LIN {X 0.147,Y -636.503,Z 756.613,A 0.000,B 0.000,C 90.000,E1 326.373} C_DIS
LIN {X -0.093,Y -640.964,Z 756.608,A 0.000,B 0.000,C 90.000,E1 325.515} C_DIS
LIN {X 0.327,Y -642.816,Z 756.606,A 0.000,B 0.000,C 90.000,E1 325.102} C_DIS
LIN {X 0.141,Y -649.762,Z 756.598,A 0.000,B 0.000,C 90.000,E1 323.623} C_DIS
LIN {X 0.029,Y -652.957,Z 756.594,A 0.000,B 0.000,C 90.000,E1 322.889} C_DIS
LIN {X 0.011,Y -657.013,Z 756.588,A 0.000,B 0.000,C 90.000,E1 321.904} C_DIS
LIN {X 0.017,Y -658.915,Z 756.586,A 0.000,B 0.000,C 90.000,E1 321.412} C_DIS
LIN {X -0.068,Y -663.423,Z 756.579,A 0.000,B 0.000,C 90.000,E1 320.194} C_DIS
LIN {X -0.059,Y -666.808,Z 756.573,A 0.000,B 0.000,C 90.000,E1 319.218} C_DIS
LIN {X -0.004,Y -670.699,Z 756.567,A 0.000,B 0.000,C 90.000,E1 318.000} C_DIS
LIN {X 0.105,Y -674.291,Z 756.560,A 0.000,B 0.000,C 90.000,E1 316.782} C_DIS
LIN {X 0.210,Y -676.958,Z 756.555,A 0.000,B 0.000,C 90.000,E1 315.810} C_DIS
LIN {X -0.087,Y -679.877,Z 756.548,A 0.000,B 0.000,C 90.000,E1 314.636} C_DIS
LIN {X 0.156,Y -682.512,Z 756.541,A 0.000,B 0.000,C 90.000,E1 313.419} C_DIS
LIN {X 0.366,Y -684.591,Z 756.536,A 0.000,B 0.000,C 90.000,E1 312.447} C_DIS
LIN {X 0.133,Y -686.391,Z 756.531,A 0.000,B 0.000,C 90.000,E1 311.515} C_DIS
LIN {X 0.436,Y -688.109,Z 756.525,A 0.000,B 0.000,C 90.000,E1 310.539} C_DIS
LIN {X -0.206,Y -689.467,Z 756.520,A 0.000,B 0.000,C 90.000,E1 309.644} C_DIS
LIN {X 0.137,Y -690.705,Z 756.515,A 0.000,B 0.000,C 90.000,E1 308.669} C_DIS
LIN {X 0.306,Y -692.395,Z 756.507,A 0.000,B 0.000,C 90.000,E1 307.237} C_DIS
LIN {X -0.100,Y -693.591,Z 756.500,A 0.000,B 0.000,C 90.000,E1 306.091} C_DIS
LIN {X 0.339,Y -694.977,Z 756.491,A 0.000,B 0.000,C 90.000,E1 304.405} C_DIS
LIN {X -0.203,Y -696.089,Z 756.484,A 0.000,B 0.000,C 90.000,E1 303.038} C_DIS
LIN {X 0.137,Y -697.503,Z 756.473,A 0.000,B 0.000,C 90.000,E1 301.131} C_DIS
LIN {X -0.043,Y -698.086,Z 756.468,A 0.000,B 0.000,C 90.000,E1 300.207} C_DIS
LIN {X -0.212,Y -698.422,Z 756.463,A 0.000,B 0.000,C 90.000,E1 299.283} C_DIS
LIN {X -0.201,Y -698.977,Z 756.453,A 0.000,B 0.000,C 90.000,E1 297.641} C_DIS
LIN {X -0.156,Y -699.561,Z 756.446,A 0.000,B 0.000,C 90.000,E1 296.232} C_DIS
LIN {X -0.010,Y -700.097,Z 756.440,A 0.000,B 0.000,C 90.000,E1 295.283} C_DIS
LIN {X -0.104,Y -700.180,Z 756.438,A 0.000,B 0.000,C 90.000,E1 294.823} C_DIS
LIN {X -0.127,Y -700.106,Z 756.437,A 0.000,B 0.000,C 90.000,E1 294.591} C_DIS
LIN {X -0.226,Y -699.545,Z 756.434,A 0.000,B 0.000,C 90.000,E1 294.131} C_DIS
LIN {X -0.243,Y -698.845,Z 756.433,A 0.000,B 0.000,C 90.000,E1 293.898} C_DIS
LIN {X 0.285,Y -696.516,Z 756.430,A 0.000,B 0.000,C 90.000,E1 293.387} C_DIS
LIN {X 0.138,Y -695.765,Z 756.429,A 0.000,B 0.000,C 90.000,E1 293.281} C_DIS
LIN {X -0.372,Y -694.648,Z 756.429,A 0.000,B 0.000,C 90.000,E1 293.206} C_DIS
LIN {X -0.246,Y -693.025,Z 756.428,A 0.000,B 0.000,C 90.000,E1 293.078} C_DIS
LIN {X -0.175,Y -688.248,Z 756.426,A 0.000,B 0.000,C 90.000,E1 292.770} C_DIS
LIN {X 0.245,Y -686.538,Z 756.426,A 0.000,B 0.000,C 90.000,E1 292.642} C_DIS
LIN {X -0.233,Y -683.886,Z 756.425,A 0.000,B 0.000,C 90.000,E1 292.589} C_DIS
LIN {X 0.315,Y -675.779,Z 756.424,A 0.000,B 0.000,C 90.000,E1 292.333} C_DIS
LIN {X -0.189,Y -668.158,Z 756.424,A 0.000,B 0.000,C 90.000,E1 292.259} C_DIS
LIN {X 0.079,Y -654.886,Z 756.423,A 0.000,B 0.000,C 90.000,E1 292.078} C_DIS
LIN {X 0.379,Y -645.016,Z 756.422,A 0.000,B 0.000,C 90.000,E1 291.897} C_DIS
LIN {X -0.041,Y -631.843,Z 756.420,A 0.000,B 0.000,C 90.000,E1 291.663} C_DIS
LIN {X 0.053,Y -611.303,Z 756.418,A 0.000,B 0.000,C 90.000,E1 291.153} C_DIS
LIN {X 0.063,Y -576.468,Z 756.412,A 0.000,B 0.000,C 90.000,E1 290.174} C_DIS
LIN {X 0.005,Y -565.947,Z 756.411,A 0.000,B 0.000,C 90.000,E1 289.885} C_DIS
LIN {X 0.011,Y -560.723,Z 756.409,A 0.000,B 0.000,C 90.000,E1 289.685} C_DIS
LIN {X 0.106,Y -557.840,Z 756.409,A 0.000,B 0.000,C 90.000,E1 289.523} C_DIS
LIN {X 0.033,Y -555.917,Z 756.407,A 0.000,B 0.000,C 90.000,E1 289.322} C_DIS
LIN {X -0.009,Y -555.886,Z 756.407,A 0.000,B 0.000,C 90.000,E1 289.322} C_DIS
LIN {X -0.098,Y -555.156,Z 756.406,A 0.000,B 0.000,C 90.000,E1 289.033} C_DIS
LIN {X -0.207,Y -554.525,Z 756.397,A 0.000,B 0.000,C 90.000,E1 287.511} C_DIS
LIN {X -0.264,Y -553.899,Z 756.388,A 0.000,B 0.000,C 90.000,E1 285.843} C_DIS
LIN {X -0.218,Y -553.135,Z 756.377,A 0.000,B 0.000,C 90.000,E1 283.883} C_DIS
LIN {X -0.030,Y -552.617,Z 756.368,A 0.000,B 0.000,C 90.000,E1 282.187} C_DIS
LIN {X 0.034,Y -552.142,Z 756.360,A 0.000,B 0.000,C 90.000,E1 280.782} C_DIS
LIN {X 0.079,Y -551.632,Z 756.352,A 0.000,B 0.000,C 90.000,E1 279.378} C_DIS
LIN {X 0.152,Y -550.794,Z 756.341,A 0.000,B 0.000,C 90.000,E1 277.409} C_DIS
LIN {X -0.212,Y -550.461,Z 756.337,A 0.000,B 0.000,C 90.000,E1 276.606} C_DIS
LIN {X 0.173,Y -549.687,Z 756.329,A 0.000,B 0.000,C 90.000,E1 275.163} C_DIS
LIN {X -0.060,Y -548.779,Z 756.321,A 0.000,B 0.000,C 90.000,E1 273.784} C_DIS
LIN {X 0.253,Y -547.842,Z 756.312,A 0.000,B 0.000,C 90.000,E1 272.064} C_DIS
LIN {X -0.045,Y -547.113,Z 756.304,A 0.000,B 0.000,C 90.000,E1 270.688} C_DIS
LIN {X 0.178,Y -546.162,Z 756.296,A 0.000,B 0.000,C 90.000,E1 269.255} C_DIS
LIN {X -0.076,Y -544.884,Z 756.285,A 0.000,B 0.000,C 90.000,E1 267.306} C_DIS
LIN {X 0.177,Y -543.801,Z 756.276,A 0.000,B 0.000,C 90.000,E1 265.584} C_DIS
LIN {X -0.176,Y -543.100,Z 756.269,A 0.000,B 0.000,C 90.000,E1 264.489} C_DIS
LIN {X 0.013,Y -542.093,Z 756.261,A 0.000,B 0.000,C 90.000,E1 263.053} C_DIS
LIN {X 0.238,Y -541.174,Z 756.255,A 0.000,B 0.000,C 90.000,E1 261.894} C_DIS
LIN {X -0.009,Y -539.986,Z 756.247,A 0.000,B 0.000,C 90.000,E1 260.500} C_DIS
LIN {X -0.206,Y -538.592,Z 756.238,A 0.000,B 0.000,C 90.000,E1 258.814} C_DIS
LIN {X 0.126,Y -537.404,Z 756.230,A 0.000,B 0.000,C 90.000,E1 257.353} C_DIS
LIN {X 0.029,Y -536.138,Z 756.222,A 0.000,B 0.000,C 90.000,E1 255.936} C_DIS
LIN {X 0.142,Y -533.945,Z 756.211,A 0.000,B 0.000,C 90.000,E1 253.921} C_DIS
LIN {X 0.017,Y -531.364,Z 756.198,A 0.000,B 0.000,C 90.000,E1 251.638} C_DIS
LIN {X -0.077,Y -529.946,Z 756.192,A 0.000,B 0.000,C 90.000,E1 250.496} C_DIS
LIN {X -0.151,Y -527.545,Z 756.182,A 0.000,B 0.000,C 90.000,E1 248.773} C_DIS
LIN {X -0.129,Y -525.940,Z 756.176,A 0.000,B 0.000,C 90.000,E1 247.614} C_DIS
LIN {X 0.280,Y -522.865,Z 756.164,A 0.000,B 0.000,C 90.000,E1 245.537} C_DIS
LIN {X -0.003,Y -519.951,Z 756.155,A 0.000,B 0.000,C 90.000,E1 243.819} C_DIS
LIN {X -0.147,Y -517.916,Z 756.148,A 0.000,B 0.000,C 90.000,E1 242.666} C_DIS
LIN {X 0.143,Y -514.638,Z 756.138,A 0.000,B 0.000,C 90.000,E1 240.873} C_DIS
LIN {X 0.053,Y -511.771,Z 756.130,A 0.000,B 0.000,C 90.000,E1 239.410} C_DIS
LIN {X 0.181,Y -508.988,Z 756.122,A 0.000,B 0.000,C 90.000,E1 237.916} C_DIS
LIN {X -0.124,Y -505.228,Z 756.112,A 0.000,B 0.000,C 90.000,E1 236.167} C_DIS
LIN {X -0.256,Y -501.763,Z 756.104,A 0.000,B 0.000,C 90.000,E1 234.689} C_DIS
LIN {X -0.081,Y -500.362,Z 756.100,A 0.000,B 0.000,C 90.000,E1 234.069} C_DIS
LIN {X -0.139,Y -495.801,Z 756.090,A 0.000,B 0.000,C 90.000,E1 232.271} C_DIS
LIN {X -0.149,Y -489.119,Z 756.075,A 0.000,B 0.000,C 90.000,E1 229.542} C_DIS
LIN {X 0.071,Y -483.618,Z 756.062,A 0.000,B 0.000,C 90.000,E1 227.067} C_DIS
LIN {X -0.269,Y -480.322,Z 756.053,A 0.000,B 0.000,C 90.000,E1 225.567} C_DIS
LIN {X -0.109,Y -475.802,Z 756.041,A 0.000,B 0.000,C 90.000,E1 223.380} C_DIS
LIN {X -0.246,Y -472.421,Z 756.032,A 0.000,B 0.000,C 90.000,E1 221.838} C_DIS
LIN {X 0.175,Y -466.911,Z 756.018,A 0.000,B 0.000,C 90.000,E1 219.277} C_DIS
LIN {X 0.169,Y -464.108,Z 756.011,A 0.000,B 0.000,C 90.000,E1 218.016} C_DIS
LIN {X -0.049,Y -460.816,Z 756.003,A 0.000,B 0.000,C 90.000,E1 216.457} C_DIS
LIN {X 0.050,Y -456.963,Z 755.992,A 0.000,B 0.000,C 90.000,E1 214.532} C_DIS
LIN {X -0.085,Y -453.088,Z 755.981,A 0.000,B 0.000,C 90.000,E1 212.625} C_DIS
LIN {X 0.080,Y -449.438,Z 755.971,A 0.000,B 0.000,C 90.000,E1 210.669} C_DIS
LIN {X -0.077,Y -445.738,Z 755.960,A 0.000,B 0.000,C 90.000,E1 208.743} C_DIS
LIN {X -0.198,Y -442.769,Z 755.951,A 0.000,B 0.000,C 90.000,E1 207.129} C_DIS
LIN {X -0.142,Y -439.022,Z 755.940,A 0.000,B 0.000,C 90.000,E1 205.155} C_DIS
LIN {X -0.189,Y -435.945,Z 755.931,A 0.000,B 0.000,C 90.000,E1 203.515} C_DIS
LIN {X -0.071,Y -432.855,Z 755.921,A 0.000,B 0.000,C 90.000,E1 201.844} C_DIS
LIN {X -0.050,Y -430.987,Z 755.916,A 0.000,B 0.000,C 90.000,E1 200.844} C_DIS
LIN {X -0.128,Y -427.203,Z 755.905,A 0.000,B 0.000,C 90.000,E1 198.852} C_DIS
LIN {X 0.121,Y -423.349,Z 755.893,A 0.000,B 0.000,C 90.000,E1 196.804} C_DIS
LIN {X -0.085,Y -420.687,Z 755.886,A 0.000,B 0.000,C 90.000,E1 195.481} C_DIS
LIN {X -0.140,Y -415.555,Z 755.871,A 0.000,B 0.000,C 90.000,E1 192.771} C_DIS
LIN {X -0.110,Y -411.974,Z 755.859,A 0.000,B 0.000,C 90.000,E1 190.715} C_DIS
LIN {X 0.023,Y -409.676,Z 755.852,A 0.000,B 0.000,C 90.000,E1 189.321} C_DIS
LIN {X 0.106,Y -405.567,Z 755.838,A 0.000,B 0.000,C 90.000,E1 186.891} C_DIS
LIN {X -0.010,Y -402.279,Z 755.827,A 0.000,B 0.000,C 90.000,E1 184.821} C_DIS
LIN {X 0.198,Y -399.205,Z 755.815,A 0.000,B 0.000,C 90.000,E1 182.694} C_DIS
LIN {X -0.027,Y -394.363,Z 755.794,A 0.000,B 0.000,C 90.000,E1 178.854} C_DIS
LIN {X 0.021,Y -392.402,Z 755.784,A 0.000,B 0.000,C 90.000,E1 177.078} C_DIS
LIN {X 0.068,Y -389.132,Z 755.764,A 0.000,B 0.000,C 90.000,E1 173.514} C_DIS
LIN {X -0.148,Y -387.186,Z 755.746,A 0.000,B 0.000,C 90.000,E1 170.330} C_DIS
LIN {X 0.109,Y -386.624,Z 755.740,A 0.000,B 0.000,C 90.000,E1 169.218} C_DIS
LIN {X 0.162,Y -385.465,Z 755.726,A 0.000,B 0.000,C 90.000,E1 166.700} C_DIS
LIN {X -0.107,Y -384.258,Z 755.710,A 0.000,B 0.000,C 90.000,E1 163.866} C_DIS
LIN {X -0.011,Y -383.574,Z 755.698,A 0.000,B 0.000,C 90.000,E1 161.692} C_DIS
LIN {X 0.228,Y -382.979,Z 755.682,A 0.000,B 0.000,C 90.000,E1 158.773} C_DIS
LIN {X -0.148,Y -382.758,Z 755.668,A 0.000,B 0.000,C 90.000,E1 156.305} C_DIS
LIN {X 0.171,Y -384.184,Z 755.634,A 0.000,B 0.000,C 90.000,E1 150.127} C_DIS
LIN {X -0.166,Y -386.094,Z 755.620,A 0.000,B 0.000,C 90.000,E1 147.661} C_DIS
LIN {X 0.178,Y -388.683,Z 755.606,A 0.000,B 0.000,C 90.000,E1 145.102} C_DIS
LIN {X -0.108,Y -392.015,Z 755.594,A 0.000,B 0.000,C 90.000,E1 143.004} C_DIS
LIN {X 0.132,Y -394.257,Z 755.589,A 0.000,B 0.000,C 90.000,E1 141.904} C_DIS
LIN {X -0.247,Y -396.105,Z 755.585,A 0.000,B 0.000,C 90.000,E1 141.251} C_DIS
LIN {X -0.056,Y -398.471,Z 755.581,A 0.000,B 0.000,C 90.000,E1 140.517} C_DIS
LIN {X -0.147,Y -401.707,Z 755.577,A 0.000,B 0.000,C 90.000,E1 139.828} C_DIS
LIN {X -0.120,Y -404.720,Z 755.574,A 0.000,B 0.000,C 90.000,E1 139.299} C_DIS
LIN {X -0.159,Y -410.004,Z 755.570,A 0.000,B 0.000,C 90.000,E1 138.609} C_DIS
LIN {X 0.021,Y -414.417,Z 755.567,A 0.000,B 0.000,C 90.000,E1 138.081} C_DIS
LIN {X -0.119,Y -432.916,Z 755.557,A 0.000,B 0.000,C 90.000,E1 136.215} C_DIS
LIN {X 0.095,Y -443.026,Z 755.551,A 0.000,B 0.000,C 90.000,E1 135.162} C_DIS
LIN {X 0.235,Y -451.554,Z 755.546,A 0.000,B 0.000,C 90.000,E1 134.271} C_DIS
LIN {X 0.103,Y -457.156,Z 755.543,A 0.000,B 0.000,C 90.000,E1 133.704} C_DIS
LIN {X 0.006,Y -466.615,Z 755.537,A 0.000,B 0.000,C 90.000,E1 132.690} C_DIS
LIN {X 0.132,Y -473.306,Z 755.533,A 0.000,B 0.000,C 90.000,E1 131.919} C_DIS
LIN {X 0.078,Y -481.138,Z 755.528,A 0.000,B 0.000,C 90.000,E1 131.024} C_DIS
LIN {X 0.143,Y -488.702,Z 755.523,A 0.000,B 0.000,C 90.000,E1 130.092} C_DIS
LIN {X 0.212,Y -494.335,Z 755.519,A 0.000,B 0.000,C 90.000,E1 129.358} C_DIS
LIN {X 0.235,Y -498.823,Z 755.516,A 0.000,B 0.000,C 90.000,E1 128.749} C_DIS
LIN {X -0.021,Y -502.992,Z 755.512,A 0.000,B 0.000,C 90.000,E1 128.177} C_DIS
LIN {X -0.147,Y -507.862,Z 755.508,A 0.000,B 0.000,C 90.000,E1 127.443} C_DIS
LIN {X 0.180,Y -512.473,Z 755.504,A 0.000,B 0.000,C 90.000,E1 126.664} C_DIS
LIN {X -0.049,Y -517.616,Z 755.499,A 0.000,B 0.000,C 90.000,E1 125.804} C_DIS
LIN {X -0.174,Y -520.957,Z 755.496,A 0.000,B 0.000,C 90.000,E1 125.231} C_DIS
LIN {X 0.068,Y -526.747,Z 755.489,A 0.000,B 0.000,C 90.000,E1 124.040} C_DIS
LIN {X -0.132,Y -528.788,Z 755.487,A 0.000,B 0.000,C 90.000,E1 123.627} C_DIS
LIN {X -0.070,Y -533.855,Z 755.480,A 0.000,B 0.000,C 90.000,E1 122.467} C_DIS
LIN {X -0.221,Y -538.603,Z 755.474,A 0.000,B 0.000,C 90.000,E1 121.337} C_DIS
LIN {X -0.039,Y -540.885,Z 755.471,A 0.000,B 0.000,C 90.000,E1 120.747} C_DIS
LIN {X 0.174,Y -543.997,Z 755.466,A 0.000,B 0.000,C 90.000,E1 119.873} C_DIS
LIN {X 0.166,Y -547.869,Z 755.460,A 0.000,B 0.000,C 90.000,E1 118.743} C_DIS
LIN {X -0.056,Y -551.564,Z 755.454,A 0.000,B 0.000,C 90.000,E1 117.641} C_DIS
LIN {X -0.028,Y -553.257,Z 755.450,A 0.000,B 0.000,C 90.000,E1 117.078} C_DIS
LIN {X 0.046,Y -555.527,Z 755.446,A 0.000,B 0.000,C 90.000,E1 116.232} C_DIS
LIN {X -0.105,Y -557.466,Z 755.441,A 0.000,B 0.000,C 90.000,E1 115.412} C_DIS
LIN {X -0.023,Y -558.612,Z 755.438,A 0.000,B 0.000,C 90.000,E1 114.847} C_DIS
LIN {X -0.137,Y -560.072,Z 755.433,A 0.000,B 0.000,C 90.000,E1 114.027} C_DIS
LIN {X -0.131,Y -562.122,Z 755.426,A 0.000,B 0.000,C 90.000,E1 112.642} C_DIS
LIN {X 0.211,Y -563.976,Z 755.418,A 0.000,B 0.000,C 90.000,E1 111.227} C_DIS
LIN {X -0.137,Y -565.743,Z 755.410,A 0.000,B 0.000,C 90.000,E1 109.885} C_DIS
LIN {X 0.080,Y -567.346,Z 755.403,A 0.000,B 0.000,C 90.000,E1 108.489} C_DIS
LIN {X -0.015,Y -568.497,Z 755.397,A 0.000,B 0.000,C 90.000,E1 107.402} C_DIS
LIN {X 0.071,Y -569.901,Z 755.389,A 0.000,B 0.000,C 90.000,E1 106.024} C_DIS
LIN {X -0.195,Y -571.583,Z 755.380,A 0.000,B 0.000,C 90.000,E1 104.411} C_DIS
LIN {X 0.043,Y -573.499,Z 755.369,A 0.000,B 0.000,C 90.000,E1 102.479} C_DIS
LIN {X 0.134,Y -575.210,Z 755.360,A 0.000,B 0.000,C 90.000,E1 100.838} C_DIS
LIN {X 0.150,Y -576.827,Z 755.351,A 0.000,B 0.000,C 90.000,E1 99.208} C_DIS
LIN {X 0.124,Y -577.570,Z 755.347,A 0.000,B 0.000,C 90.000,E1 98.398} C_DIS
LIN {X 0.097,Y -578.942,Z 755.338,A 0.000,B 0.000,C 90.000,E1 96.777} C_DIS
LIN {X 0.237,Y -579.878,Z 755.332,A 0.000,B 0.000,C 90.000,E1 95.682} C_DIS
LIN {X -0.030,Y -580.869,Z 755.324,A 0.000,B 0.000,C 90.000,E1 94.359} C_DIS
LIN {X -0.118,Y -581.978,Z 755.315,A 0.000,B 0.000,C 90.000,E1 92.751} C_DIS
LIN {X -0.216,Y -582.998,Z 755.306,A 0.000,B 0.000,C 90.000,E1 91.146} C_DIS
LIN {X 0.099,Y -583.679,Z 755.299,A 0.000,B 0.000,C 90.000,E1 89.771} C_DIS
LIN {X -0.161,Y -584.225,Z 755.291,A 0.000,B 0.000,C 90.000,E1 88.453} C_DIS
LIN {X 0.184,Y -584.671,Z 755.284,A 0.000,B 0.000,C 90.000,E1 87.078} C_DIS
LIN {X -0.229,Y -584.996,Z 755.278,A 0.000,B 0.000,C 90.000,E1 86.045} C_DIS
LIN {X -0.014,Y -585.341,Z 755.268,A 0.000,B 0.000,C 90.000,E1 84.147} C_DIS
LIN {X -0.132,Y -585.461,Z 755.260,A 0.000,B 0.000,C 90.000,E1 82.818} C_DIS
LIN {X -0.001,Y -585.518,Z 755.251,A 0.000,B 0.000,C 90.000,E1 81.197} C_DIS
LIN {X -0.021,Y -585.419,Z 755.244,A 0.000,B 0.000,C 90.000,E1 79.859} C_DIS
LIN {X -0.130,Y -585.006,Z 755.233,A 0.000,B 0.000,C 90.000,E1 77.993} C_DIS
LIN {X 0.276,Y -584.665,Z 755.227,A 0.000,B 0.000,C 90.000,E1 76.881} C_DIS
LIN {X -0.083,Y -584.186,Z 755.220,A 0.000,B 0.000,C 90.000,E1 75.574} C_DIS
LIN {X -0.211,Y -583.403,Z 755.211,A 0.000,B 0.000,C 90.000,E1 73.976} C_DIS
LIN {X -0.259,Y -582.865,Z 755.205,A 0.000,B 0.000,C 90.000,E1 72.906} C_DIS
LIN {X -0.144,Y -582.196,Z 755.199,A 0.000,B 0.000,C 90.000,E1 71.819} C_DIS
LIN {X -0.037,Y -581.479,Z 755.193,A 0.000,B 0.000,C 90.000,E1 70.732} C_DIS
LIN {X 0.053,Y -580.686,Z 755.187,A 0.000,B 0.000,C 90.000,E1 69.645} C_DIS
LIN {X -0.209,Y -579.834,Z 755.181,A 0.000,B 0.000,C 90.000,E1 68.592} C_DIS
LIN {X 0.297,Y -578.313,Z 755.172,A 0.000,B 0.000,C 90.000,E1 66.922} C_DIS
LIN {X 0.002,Y -577.115,Z 755.166,A 0.000,B 0.000,C 90.000,E1 65.869} C_DIS
LIN {X -0.227,Y -575.426,Z 755.158,A 0.000,B 0.000,C 90.000,E1 64.537} C_DIS
LIN {X -0.070,Y -573.908,Z 755.152,A 0.000,B 0.000,C 90.000,E1 63.435} C_DIS
LIN {X -0.192,Y -572.092,Z 755.146,A 0.000,B 0.000,C 90.000,E1 62.359} C_DIS
LIN {X 0.254,Y -571.151,Z 755.143,A 0.000,B 0.000,C 90.000,E1 61.769} C_DIS
LIN {X 0.023,Y -569.534,Z 755.139,A 0.000,B 0.000,C 90.000,E1 60.973} C_DIS
LIN {X 0.095,Y -567.059,Z 755.133,A 0.000,B 0.000,C 90.000,E1 59.871} C_DIS
LIN {X -0.176,Y -565.009,Z 755.128,A 0.000,B 0.000,C 90.000,E1 59.076} C_DIS
LIN {X 0.104,Y -561.994,Z 755.122,A 0.000,B 0.000,C 90.000,E1 57.946} C_DIS
LIN {X 0.074,Y -559.449,Z 755.117,A 0.000,B 0.000,C 90.000,E1 57.120} C_DIS
LIN {X 0.022,Y -556.695,Z 755.113,A 0.000,B 0.000,C 90.000,E1 56.294} C_DIS
LIN {X -0.058,Y -553.679,Z 755.108,A 0.000,B 0.000,C 90.000,E1 55.468} C_DIS
LIN {X 0.080,Y -551.539,Z 755.105,A 0.000,B 0.000,C 90.000,E1 54.895} C_DIS
LIN {X -0.058,Y -547.862,Z 755.100,A 0.000,B 0.000,C 90.000,E1 54.069} C_DIS
LIN {X 0.220,Y -544.487,Z 755.096,A 0.000,B 0.000,C 90.000,E1 53.336} C_DIS
LIN {X 0.142,Y -540.806,Z 755.093,A 0.000,B 0.000,C 90.000,E1 52.637} C_DIS
LIN {X 0.184,Y -537.677,Z 755.089,A 0.000,B 0.000,C 90.000,E1 52.065} C_DIS
LIN {X -0.218,Y -534.241,Z 755.086,A 0.000,B 0.000,C 90.000,E1 51.537} C_DIS
LIN {X 0.111,Y -530.399,Z 755.083,A 0.000,B 0.000,C 90.000,E1 50.928} C_DIS
LIN {X 0.076,Y -526.160,Z 755.080,A 0.000,B 0.000,C 90.000,E1 50.356} C_DIS
LIN {X 0.005,Y -521.419,Z 755.077,A 0.000,B 0.000,C 90.000,E1 49.784} C_DIS
LIN {X -0.287,Y -517.500,Z 755.074,A 0.000,B 0.000,C 90.000,E1 49.380} C_DIS
LIN {X 0.141,Y -511.949,Z 755.071,A 0.000,B 0.000,C 90.000,E1 48.771} C_DIS
LIN {X 0.147,Y -506.064,Z 755.068,A 0.000,B 0.000,C 90.000,E1 48.243} C_DIS
LIN {X -0.011,Y -500.020,Z 755.065,A 0.000,B 0.000,C 90.000,E1 47.757} C_DIS
LIN {X -0.004,Y -495.364,Z 755.063,A 0.000,B 0.000,C 90.000,E1 47.391} C_DIS
LIN {X 0.092,Y -485.900,Z 755.060,A 0.000,B 0.000,C 90.000,E1 46.701} C_DIS
LIN {X 0.283,Y -477.589,Z 755.057,A 0.000,B 0.000,C 90.000,E1 46.134} C_DIS
LIN {X 0.055,Y -464.629,Z 755.052,A 0.000,B 0.000,C 90.000,E1 45.324} C_DIS
LIN {X -0.039,Y -448.446,Z 755.046,A 0.000,B 0.000,C 90.000,E1 44.271} C_DIS
LIN {X -0.168,Y -430.904,Z 755.039,A 0.000,B 0.000,C 90.000,E1 43.095} C_DIS
LIN {X -0.150,Y -418.349,Z 755.034,A 0.000,B 0.000,C 90.000,E1 42.162} C_DIS
LIN {X 0.173,Y -411.321,Z 755.031,A 0.000,B 0.000,C 90.000,E1 41.515} C_DIS
LIN {X 0.148,Y -411.287,Z 755.031,A 0.000,B 0.000,C 90.000,E1 41.515} C_DIS
LIN {X 0.128,Y -406.117,Z 755.015,A 0.000,B 0.000,C 90.000,E1 38.624} C_DIS
LIN {X 0.094,Y -404.663,Z 755.011,A 0.000,B 0.000,C 90.000,E1 37.935} C_DIS
LIN {X 0.157,Y -400.734,Z 755.000,A 0.000,B 0.000,C 90.000,E1 36.011} C_DIS
LIN {X 0.034,Y -401.288,Z 754.982,A 0.000,B 0.000,C 90.000,E1 32.704} C_DIS
LIN {X 0.150,Y -402.061,Z 754.970,A 0.000,B 0.000,C 90.000,E1 30.590} C_DIS
LIN {X 0.213,Y -403.125,Z 754.958,A 0.000,B 0.000,C 90.000,E1 28.487} C_DIS
LIN {X -0.179,Y -404.455,Z 754.945,A 0.000,B 0.000,C 90.000,E1 26.104} C_DIS
LIN {X -0.255,Y -406.401,Z 754.930,A 0.000,B 0.000,C 90.000,E1 23.334} C_DIS
LIN {X -0.088,Y -409.961,Z 754.908,A 0.000,B 0.000,C 90.000,E1 19.504} C_DIS
LIN {X 0.062,Y -413.764,Z 754.891,A 0.000,B 0.000,C 90.000,E1 16.386} C_DIS
LIN {X -0.059,Y -417.194,Z 754.878,A 0.000,B 0.000,C 90.000,E1 14.008} C_DIS
LIN {X 0.060,Y -420.404,Z 754.867,A 0.000,B 0.000,C 90.000,E1 11.951} C_DIS
LIN {X 0.088,Y -423.115,Z 754.857,A 0.000,B 0.000,C 90.000,E1 10.254} C_DIS
LIN {X 0.178,Y -426.402,Z 754.846,A 0.000,B 0.000,C 90.000,E1 8.219} C_DIS
LIN {X -0.199,Y -429.689,Z 754.835,A 0.000,B 0.000,C 90.000,E1 6.258} C_DIS
LIN {X 0.167,Y -434.933,Z 754.818,A 0.000,B 0.000,C 90.000,E1 3.212} C_DIS
LIN {X 0.020,Y -439.251,Z 754.805,A 0.000,B 0.000,C 90.000,E1 0.917} C_DIS
LIN {X 0.093,Y -443.383,Z 754.793,A 0.000,B 0.000,C 90.000,E1 358.797} C_DIS
LIN {X 0.180,Y -448.205,Z 754.781,A 0.000,B 0.000,C 90.000,E1 356.502} C_DIS
LIN {X -0.110,Y -454.722,Z 754.765,A 0.000,B 0.000,C 90.000,E1 353.628} C_DIS
LIN {X 0.017,Y -458.414,Z 754.756,A 0.000,B 0.000,C 90.000,E1 352.008} C_DIS
LIN {X 0.218,Y -461.862,Z 754.747,A 0.000,B 0.000,C 90.000,E1 350.387} C_DIS
LIN {X 0.051,Y -463.825,Z 754.742,A 0.000,B 0.000,C 90.000,E1 349.454} C_DIS
LIN {X -0.029,Y -466.937,Z 754.733,A 0.000,B 0.000,C 90.000,E1 347.881} C_DIS
LIN {X -0.033,Y -470.469,Z 754.722,A 0.000,B 0.000,C 90.000,E1 345.992} C_DIS
LIN {X -0.181,Y -473.157,Z 754.715,A 0.000,B 0.000,C 90.000,E1 344.755} C_DIS
LIN {X 0.049,Y -475.010,Z 754.712,A 0.000,B 0.000,C 90.000,E1 344.102} C_DIS
LIN {X 0.082,Y -476.722,Z 754.709,A 0.000,B 0.000,C 90.000,E1 343.630} C_DIS
LIN {X -0.155,Y -478.581,Z 754.707,A 0.000,B 0.000,C 90.000,E1 343.268} C_DIS
LIN {X 0.038,Y -481.411,Z 754.704,A 0.000,B 0.000,C 90.000,E1 342.779} C_DIS
LIN {X -0.237,Y -485.394,Z 754.702,A 0.000,B 0.000,C 90.000,E1 342.308} C_DIS
LIN {X 0.242,Y -489.667,Z 754.699,A 0.000,B 0.000,C 90.000,E1 341.819} C_DIS
LIN {X -0.158,Y -493.067,Z 754.698,A 0.000,B 0.000,C 90.000,E1 341.583} C_DIS
LIN {X -0.018,Y -505.279,Z 754.693,A 0.000,B 0.000,C 90.000,E1 340.678} C_DIS
LIN {X -0.201,Y -519.557,Z 754.687,A 0.000,B 0.000,C 90.000,E1 339.752} C_DIS
LIN {X -0.138,Y -535.697,Z 754.682,A 0.000,B 0.000,C 90.000,E1 338.773} C_DIS
LIN {X 0.025,Y -540.483,Z 754.680,A 0.000,B 0.000,C 90.000,E1 338.465} C_DIS
LIN {X 0.080,Y -546.277,Z 754.678,A 0.000,B 0.000,C 90.000,E1 338.050} C_DIS
LIN {X 0.017,Y -552.136,Z 754.676,A 0.000,B 0.000,C 90.000,E1 337.614} C_DIS
LIN {X -0.106,Y -556.162,Z 754.674,A 0.000,B 0.000,C 90.000,E1 337.283} C_DIS
LIN {X -0.127,Y -561.410,Z 754.671,A 0.000,B 0.000,C 90.000,E1 336.794} C_DIS
LIN {X -0.356,Y -567.575,Z 754.667,A 0.000,B 0.000,C 90.000,E1 336.177} C_DIS
LIN {X -0.134,Y -572.458,Z 754.664,A 0.000,B 0.000,C 90.000,E1 335.613} C_DIS
LIN {X -0.019,Y -578.287,Z 754.661,A 0.000,B 0.000,C 90.000,E1 334.921} C_DIS
LIN {X 0.014,Y -585.920,Z 754.655,A 0.000,B 0.000,C 90.000,E1 333.973} C_DIS
LIN {X -0.122,Y -593.044,Z 754.650,A 0.000,B 0.000,C 90.000,E1 333.050} C_DIS
LIN {X 0.130,Y -598.901,Z 754.646,A 0.000,B 0.000,C 90.000,E1 332.231} C_DIS
LIN {X 0.160,Y -605.428,Z 754.641,A 0.000,B 0.000,C 90.000,E1 331.307} C_DIS
LIN {X -0.025,Y -611.666,Z 754.636,A 0.000,B 0.000,C 90.000,E1 330.411} C_DIS
LIN {X -0.388,Y -618.403,Z 754.630,A 0.000,B 0.000,C 90.000,E1 329.410} C_DIS
LIN {X 0.198,Y -623.921,Z 754.625,A 0.000,B 0.000,C 90.000,E1 328.456} C_DIS
LIN {X -0.002,Y -629.239,Z 754.620,A 0.000,B 0.000,C 90.000,E1 327.582} C_DIS
LIN {X 0.072,Y -634.726,Z 754.614,A 0.000,B 0.000,C 90.000,E1 326.580} C_DIS
LIN {X -0.178,Y -639.919,Z 754.609,A 0.000,B 0.000,C 90.000,E1 325.595} C_DIS
LIN {X -0.336,Y -645.369,Z 754.603,A 0.000,B 0.000,C 90.000,E1 324.482} C_DIS
LIN {X -0.064,Y -650.005,Z 754.597,A 0.000,B 0.000,C 90.000,E1 323.463} C_DIS
LIN {X -0.096,Y -652.160,Z 754.594,A 0.000,B 0.000,C 90.000,E1 322.970} C_DIS
LIN {X -0.183,Y -657.246,Z 754.587,A 0.000,B 0.000,C 90.000,E1 321.743} C_DIS
LIN {X -0.197,Y -661.905,Z 754.581,A 0.000,B 0.000,C 90.000,E1 320.517} C_DIS
LIN {X -0.213,Y -665.409,Z 754.575,A 0.000,B 0.000,C 90.000,E1 319.542} C_DIS
LIN {X -0.185,Y -668.643,Z 754.570,A 0.000,B 0.000,C 90.000,E1 318.566} C_DIS
LIN {X 0.329,Y -671.666,Z 754.564,A 0.000,B 0.000,C 90.000,E1 317.553} C_DIS
LIN {X -0.064,Y -674.546,Z 754.559,A 0.000,B 0.000,C 90.000,E1 316.620} C_DIS
LIN {X 0.046,Y -677.229,Z 754.554,A 0.000,B 0.000,C 90.000,E1 315.648} C_DIS
LIN {X 0.234,Y -680.181,Z 754.547,A 0.000,B 0.000,C 90.000,E1 314.433} C_DIS
LIN {X 0.051,Y -683.365,Z 754.539,A 0.000,B 0.000,C 90.000,E1 313.014} C_DIS
LIN {X 0.211,Y -684.880,Z 754.535,A 0.000,B 0.000,C 90.000,E1 312.285} C_DIS
LIN {X -0.079,Y -686.279,Z 754.531,A 0.000,B 0.000,C 90.000,E1 311.595} C_DIS
LIN {X 0.284,Y -688.406,Z 754.524,A 0.000,B 0.000,C 90.000,E1 310.378} C_DIS
LIN {X 0.237,Y -690.129,Z 754.518,A 0.000,B 0.000,C 90.000,E1 309.197} C_DIS
LIN {X -0.148,Y -691.885,Z 754.510,A 0.000,B 0.000,C 90.000,E1 307.810} C_DIS
LIN {X -0.205,Y -692.986,Z 754.505,A 0.000,B 0.000,C 90.000,E1 306.870} C_DIS
LIN {X -0.253,Y -693.846,Z 754.500,A 0.000,B 0.000,C 90.000,E1 305.931} C_DIS
LIN {X 0.139,Y -695.069,Z 754.492,A 0.000,B 0.000,C 90.000,E1 304.485} C_DIS
LIN {X -0.017,Y -696.187,Z 754.484,A 0.000,B 0.000,C 90.000,E1 303.086} C_DIS
LIN {X -0.298,Y -697.410,Z 754.475,A 0.000,B 0.000,C 90.000,E1 301.465} C_DIS
LIN {X -0.125,Y -698.095,Z 754.469,A 0.000,B 0.000,C 90.000,E1 300.512} C_DIS
LIN {X 0.303,Y -698.461,Z 754.464,A 0.000,B 0.000,C 90.000,E1 299.539} C_DIS
LIN {X 0.049,Y -698.940,Z 754.456,A 0.000,B 0.000,C 90.000,E1 298.153} C_DIS
LIN {X 0.001,Y -699.648,Z 754.446,A 0.000,B 0.000,C 90.000,E1 296.283} C_DIS
LIN {X 0.116,Y -700.236,Z 754.440,A 0.000,B 0.000,C 90.000,E1 295.103} C_DIS
LIN {X 0.023,Y -700.298,Z 754.437,A 0.000,B 0.000,C 90.000,E1 294.643} C_DIS
LIN {X -0.364,Y -699.701,Z 754.434,A 0.000,B 0.000,C 90.000,E1 294.207} C_DIS
LIN {X -0.095,Y -699.197,Z 754.433,A 0.000,B 0.000,C 90.000,E1 293.951} C_DIS
LIN {X 0.155,Y -696.837,Z 754.430,A 0.000,B 0.000,C 90.000,E1 293.462} C_DIS
LIN {X 0.284,Y -696.173,Z 754.430,A 0.000,B 0.000,C 90.000,E1 293.334} C_DIS
LIN {X -0.226,Y -695.270,Z 754.429,A 0.000,B 0.000,C 90.000,E1 293.259} C_DIS
LIN {X -0.100,Y -693.925,Z 754.429,A 0.000,B 0.000,C 90.000,E1 293.131} C_DIS
LIN {X -0.045,Y -689.105,Z 754.427,A 0.000,B 0.000,C 90.000,E1 292.823} C_DIS
LIN {X 0.123,Y -687.410,Z 754.426,A 0.000,B 0.000,C 90.000,E1 292.717} C_DIS
LIN {X -0.077,Y -685.318,Z 754.426,A 0.000,B 0.000,C 90.000,E1 292.642} C_DIS
LIN {X -0.300,Y -682.961,Z 754.425,A 0.000,B 0.000,C 90.000,E1 292.589} C_DIS
LIN {X 0.319,Y -674.786,Z 754.424,A 0.000,B 0.000,C 90.000,E1 292.333} C_DIS
LIN {X 0.352,Y -665.808,Z 754.424,A 0.000,B 0.000,C 90.000,E1 292.206} C_DIS
LIN {X -0.288,Y -656.454,Z 754.423,A 0.000,B 0.000,C 90.000,E1 292.153} C_DIS
LIN {X 0.040,Y -646.227,Z 754.422,A 0.000,B 0.000,C 90.000,E1 291.972} C_DIS
LIN {X -0.007,Y -633.401,Z 754.421,A 0.000,B 0.000,C 90.000,E1 291.716} C_DIS
LIN {X -0.054,Y -612.931,Z 754.418,A 0.000,B 0.000,C 90.000,E1 291.227} C_DIS
LIN {X 0.242,Y -585.229,Z 754.414,A 0.000,B 0.000,C 90.000,E1 290.429} C_DIS
LIN {X -0.255,Y -572.681,Z 754.412,A 0.000,B 0.000,C 90.000,E1 290.120} C_DIS
LIN {X 0.110,Y -567.261,Z 754.411,A 0.000,B 0.000,C 90.000,E1 289.939} C_DIS
LIN {X 0.044,Y -562.012,Z 754.410,A 0.000,B 0.000,C 90.000,E1 289.758} C_DIS
LIN {X -0.115,Y -558.018,Z 754.409,A 0.000,B 0.000,C 90.000,E1 289.577} C_DIS
LIN {X 0.128,Y -557.507,Z 754.409,A 0.000,B 0.000,C 90.000,E1 289.523} C_DIS
LIN {X -0.292,Y -555.973,Z 754.408,A 0.000,B 0.000,C 90.000,E1 289.396} C_DIS
LIN {X -0.334,Y -555.955,Z 754.408,A 0.000,B 0.000,C 90.000,E1 289.396} C_DIS
LIN {X 0.054,Y -555.260,Z 754.406,A 0.000,B 0.000,C 90.000,E1 289.087} C_DIS
LIN {X -0.261,Y -554.831,Z 754.403,A 0.000,B 0.000,C 90.000,E1 288.544} C_DIS
LIN {X -0.006,Y -554.456,Z 754.397,A 0.000,B 0.000,C 90.000,E1 287.402} C_DIS
LIN {X 0.095,Y -553.828,Z 754.387,A 0.000,B 0.000,C 90.000,E1 285.717} C_DIS
LIN {X -0.002,Y -553.099,Z 754.377,A 0.000,B 0.000,C 90.000,E1 283.772} C_DIS
LIN {X -0.231,Y -552.563,Z 754.367,A 0.000,B 0.000,C 90.000,E1 282.119} C_DIS
LIN {X -0.177,Y -552.111,Z 754.359,A 0.000,B 0.000,C 90.000,E1 280.715} C_DIS
LIN {X -0.234,Y -551.554,Z 754.352,A 0.000,B 0.000,C 90.000,E1 279.321} C_DIS
LIN {X 0.243,Y -550.949,Z 754.344,A 0.000,B 0.000,C 90.000,E1 277.871} C_DIS
LIN {X -0.016,Y -550.500,Z 754.338,A 0.000,B 0.000,C 90.000,E1 276.777} C_DIS
LIN {X -0.277,Y -549.940,Z 754.331,A 0.000,B 0.000,C 90.000,E1 275.682} C_DIS
LIN {X 0.045,Y -549.072,Z 754.324,A 0.000,B 0.000,C 90.000,E1 274.245} C_DIS
LIN {X -0.105,Y -547.973,Z 754.313,A 0.000,B 0.000,C 90.000,E1 272.293} C_DIS
LIN {X 0.192,Y -547.076,Z 754.303,A 0.000,B 0.000,C 90.000,E1 270.573} C_DIS
LIN {X -0.091,Y -545.958,Z 754.294,A 0.000,B 0.000,C 90.000,E1 268.912} C_DIS
LIN {X 0.190,Y -544.656,Z 754.283,A 0.000,B 0.000,C 90.000,E1 266.906} C_DIS
LIN {X -0.135,Y -543.779,Z 754.275,A 0.000,B 0.000,C 90.000,E1 265.527} C_DIS
LIN {X 0.052,Y -543.041,Z 754.269,A 0.000,B 0.000,C 90.000,E1 264.375} C_DIS
LIN {X 0.228,Y -542.256,Z 754.263,A 0.000,B 0.000,C 90.000,E1 263.223} C_DIS
LIN {X -0.153,Y -541.353,Z 754.256,A 0.000,B 0.000,C 90.000,E1 262.129} C_DIS
LIN {X 0.133,Y -540.169,Z 754.248,A 0.000,B 0.000,C 90.000,E1 260.679} C_DIS
LIN {X -0.069,Y -538.749,Z 754.239,A 0.000,B 0.000,C 90.000,E1 258.993} C_DIS
LIN {X -0.262,Y -537.583,Z 754.231,A 0.000,B 0.000,C 90.000,E1 257.589} C_DIS
LIN {X 0.163,Y -536.321,Z 754.223,A 0.000,B 0.000,C 90.000,E1 256.117} C_DIS
LIN {X -0.005,Y -535.107,Z 754.217,A 0.000,B 0.000,C 90.000,E1 254.991} C_DIS
LIN {X -0.192,Y -533.882,Z 754.210,A 0.000,B 0.000,C 90.000,E1 253.866} C_DIS
LIN {X 0.159,Y -531.606,Z 754.199,A 0.000,B 0.000,C 90.000,E1 251.819} C_DIS
LIN {X 0.069,Y -530.258,Z 754.193,A 0.000,B 0.000,C 90.000,E1 250.678} C_DIS
LIN {X 0.002,Y -527.880,Z 754.183,A 0.000,B 0.000,C 90.000,E1 248.954} C_DIS
LIN {X 0.031,Y -526.270,Z 754.177,A 0.000,B 0.000,C 90.000,E1 247.794} C_DIS
LIN {X 0.076,Y -523.619,Z 754.167,A 0.000,B 0.000,C 90.000,E1 246.049} C_DIS
LIN {X 0.075,Y -522.258,Z 754.162,A 0.000,B 0.000,C 90.000,E1 245.177} C_DIS
LIN {X 0.096,Y -519.846,Z 754.154,A 0.000,B 0.000,C 90.000,E1 243.717} C_DIS
LIN {X -0.190,Y -518.337,Z 754.149,A 0.000,B 0.000,C 90.000,E1 242.871} C_DIS
LIN {X -0.005,Y -515.628,Z 754.141,A 0.000,B 0.000,C 90.000,E1 241.385} C_DIS
LIN {X 0.020,Y -512.222,Z 754.131,A 0.000,B 0.000,C 90.000,E1 239.616} C_DIS
LIN {X -0.213,Y -508.816,Z 754.121,A 0.000,B 0.000,C 90.000,E1 237.867} C_DIS
LIN {X -0.142,Y -505.678,Z 754.113,A 0.000,B 0.000,C 90.000,E1 236.373} C_DIS
LIN {X -0.154,Y -502.958,Z 754.107,A 0.000,B 0.000,C 90.000,E1 235.182} C_DIS
LIN {X -0.203,Y -500.133,Z 754.100,A 0.000,B 0.000,C 90.000,E1 233.989} C_DIS
LIN {X -0.262,Y -495.606,Z 754.090,A 0.000,B 0.000,C 90.000,E1 232.190} C_DIS
LIN {X -0.118,Y -488.211,Z 754.073,A 0.000,B 0.000,C 90.000,E1 229.138} C_DIS
LIN {X -0.198,Y -484.099,Z 754.063,A 0.000,B 0.000,C 90.000,E1 227.310} C_DIS
LIN {X 0.152,Y -480.811,Z 754.054,A 0.000,B 0.000,C 90.000,E1 225.729} C_DIS
LIN {X 0.208,Y -476.867,Z 754.044,A 0.000,B 0.000,C 90.000,E1 223.866} C_DIS
LIN {X 0.313,Y -474.243,Z 754.037,A 0.000,B 0.000,C 90.000,E1 222.609} C_DIS
LIN {X 0.283,Y -472.259,Z 754.032,A 0.000,B 0.000,C 90.000,E1 221.676} C_DIS
LIN {X -0.030,Y -467.389,Z 754.020,A 0.000,B 0.000,C 90.000,E1 219.519} C_DIS
LIN {X -0.024,Y -464.608,Z 754.013,A 0.000,B 0.000,C 90.000,E1 218.257} C_DIS
LIN {X 0.051,Y -461.285,Z 754.004,A 0.000,B 0.000,C 90.000,E1 216.664} C_DIS
LIN {X -0.110,Y -456.755,Z 753.991,A 0.000,B 0.000,C 90.000,E1 214.452} C_DIS
LIN {X -0.154,Y -452.285,Z 753.979,A 0.000,B 0.000,C 90.000,E1 212.212} C_DIS
LIN {X -0.013,Y -448.621,Z 753.968,A 0.000,B 0.000,C 90.000,E1 210.256} C_DIS
LIN {X -0.016,Y -444.991,Z 753.957,A 0.000,B 0.000,C 90.000,E1 208.309} C_DIS
LIN {X 0.006,Y -442.617,Z 753.950,A 0.000,B 0.000,C 90.000,E1 207.001} C_DIS
LIN {X 0.057,Y -438.873,Z 753.939,A 0.000,B 0.000,C 90.000,E1 205.027} C_DIS
LIN {X 0.005,Y -435.792,Z 753.930,A 0.000,B 0.000,C 90.000,E1 203.387} C_DIS
LIN {X 0.117,Y -432.711,Z 753.921,A 0.000,B 0.000,C 90.000,E1 201.716} C_DIS
LIN {X -0.020,Y -430.823,Z 753.915,A 0.000,B 0.000,C 90.000,E1 200.737} C_DIS
LIN {X 0.048,Y -427.061,Z 753.904,A 0.000,B 0.000,C 90.000,E1 198.725} C_DIS
LIN {X -0.121,Y -423.187,Z 753.893,A 0.000,B 0.000,C 90.000,E1 196.732} C_DIS
LIN {X -0.215,Y -419.192,Z 753.882,A 0.000,B 0.000,C 90.000,E1 194.717} C_DIS
LIN {X 0.001,Y -415.444,Z 753.870,A 0.000,B 0.000,C 90.000,E1 192.647} C_DIS
LIN {X -0.057,Y -411.873,Z 753.859,A 0.000,B 0.000,C 90.000,E1 190.602} C_DIS
LIN {X 0.078,Y -409.566,Z 753.851,A 0.000,B 0.000,C 90.000,E1 189.208} C_DIS
LIN {X 0.168,Y -404.947,Z 753.836,A 0.000,B 0.000,C 90.000,E1 186.429} C_DIS
LIN {X -0.024,Y -400.699,Z 753.820,A 0.000,B 0.000,C 90.000,E1 183.669} C_DIS
LIN {X -0.114,Y -395.966,Z 753.801,A 0.000,B 0.000,C 90.000,E1 180.172} C_DIS
LIN {X -0.168,Y -393.223,Z 753.787,A 0.000,B 0.000,C 90.000,E1 177.707} C_DIS
LIN {X -0.166,Y -389.487,Z 753.765,A 0.000,B 0.000,C 90.000,E1 173.799} C_DIS
LIN {X -0.096,Y -387.163,Z 753.744,A 0.000,B 0.000,C 90.000,E1 169.859} C_DIS
LIN {X -0.094,Y -385.786,Z 753.728,A 0.000,B 0.000,C 90.000,E1 166.992} C_DIS
LIN {X 0.161,Y -385.143,Z 753.720,A 0.000,B 0.000,C 90.000,E1 165.519} C_DIS
LIN {X 0.077,Y -384.289,Z 753.706,A 0.000,B 0.000,C 90.000,E1 163.015} C_DIS
LIN {X -0.118,Y -383.392,Z 753.686,A 0.000,B 0.000,C 90.000,E1 159.444} C_DIS
LIN {X 0.034,Y -383.043,Z 753.670,A 0.000,B 0.000,C 90.000,E1 156.538} C_DIS
LIN {X -0.194,Y -382.996,Z 753.658,A 0.000,B 0.000,C 90.000,E1 154.409} C_DIS
LIN {X -0.139,Y -385.226,Z 753.628,A 0.000,B 0.000,C 90.000,E1 148.997} C_DIS
LIN {X 0.074,Y -388.916,Z 753.606,A 0.000,B 0.000,C 90.000,E1 145.022} C_DIS
LIN {X -0.205,Y -392.129,Z 753.594,A 0.000,B 0.000,C 90.000,E1 142.924} C_DIS
LIN {X 0.037,Y -394.320,Z 753.588,A 0.000,B 0.000,C 90.000,E1 141.823} C_DIS
LIN {X -0.139,Y -396.639,Z 753.583,A 0.000,B 0.000,C 90.000,E1 140.964} C_DIS
LIN {X -0.147,Y -398.438,Z 753.580,A 0.000,B 0.000,C 90.000,E1 140.436} C_DIS
LIN {X 0.065,Y -401.530,Z 753.576,A 0.000,B 0.000,C 90.000,E1 139.703} C_DIS
LIN {X 0.162,Y -404.159,Z 753.574,A 0.000,B 0.000,C 90.000,E1 139.218} C_DIS
LIN {X 0.066,Y -408.240,Z 753.570,A 0.000,B 0.000,C 90.000,E1 138.647} C_DIS
LIN {X -0.188,Y -413.330,Z 753.567,A 0.000,B 0.000,C 90.000,E1 138.081} C_DIS
LIN {X 0.121,Y -425.127,Z 753.560,A 0.000,B 0.000,C 90.000,E1 136.824} C_DIS
LIN {X -0.004,Y -433.841,Z 753.555,A 0.000,B 0.000,C 90.000,E1 135.972} C_DIS
LIN {X -0.009,Y -445.402,Z 753.549,A 0.000,B 0.000,C 90.000,E1 134.798} C_DIS
LIN {X 0.042,Y -456.798,Z 753.542,A 0.000,B 0.000,C 90.000,E1 133.623} C_DIS
LIN {X -0.177,Y -466.470,Z 753.537,A 0.000,B 0.000,C 90.000,E1 132.609} C_DIS
LIN {X -0.080,Y -471.876,Z 753.533,A 0.000,B 0.000,C 90.000,E1 132.000} C_DIS
LIN {X 0.097,Y -479.939,Z 753.528,A 0.000,B 0.000,C 90.000,E1 131.067} C_DIS
LIN {X -0.015,Y -488.809,Z 753.522,A 0.000,B 0.000,C 90.000,E1 130.011} C_DIS
LIN {X -0.270,Y -494.774,Z 753.518,A 0.000,B 0.000,C 90.000,E1 129.277} C_DIS
LIN {X -0.005,Y -499.067,Z 753.515,A 0.000,B 0.000,C 90.000,E1 128.669} C_DIS
LIN {X -0.243,Y -503.228,Z 753.512,A 0.000,B 0.000,C 90.000,E1 128.096} C_DIS
LIN {X -0.188,Y -507.006,Z 753.508,A 0.000,B 0.000,C 90.000,E1 127.523} C_DIS
LIN {X -0.057,Y -510.781,Z 753.505,A 0.000,B 0.000,C 90.000,E1 126.916} C_DIS
LIN {X 0.183,Y -514.358,Z 753.502,A 0.000,B 0.000,C 90.000,E1 126.297} C_DIS
LIN {X -0.040,Y -520.198,Z 753.496,A 0.000,B 0.000,C 90.000,E1 125.311} C_DIS
LIN {X -0.097,Y -521.757,Z 753.495,A 0.000,B 0.000,C 90.000,E1 125.025} C_DIS
LIN {X -0.134,Y -527.534,Z 753.488,A 0.000,B 0.000,C 90.000,E1 123.865} C_DIS
LIN {X 0.205,Y -532.650,Z 753.482,A 0.000,B 0.000,C 90.000,E1 122.673} C_DIS
LIN {X 0.331,Y -536.360,Z 753.477,A 0.000,B 0.000,C 90.000,E1 121.799} C_DIS
LIN {X -0.107,Y -540.450,Z 753.471,A 0.000,B 0.000,C 90.000,E1 120.846} C_DIS
LIN {X -0.179,Y -543.612,Z 753.467,A 0.000,B 0.000,C 90.000,E1 120.001} C_DIS
LIN {X -0.196,Y -547.536,Z 753.460,A 0.000,B 0.000,C 90.000,E1 118.871} C_DIS
LIN {X 0.062,Y -551.244,Z 753.454,A 0.000,B 0.000,C 90.000,E1 117.719} C_DIS
LIN {X 0.115,Y -553.818,Z 753.449,A 0.000,B 0.000,C 90.000,E1 116.873} C_DIS
LIN {X -0.054,Y -556.045,Z 753.445,A 0.000,B 0.000,C 90.000,E1 116.052} C_DIS
LIN {X 0.042,Y -557.945,Z 753.440,A 0.000,B 0.000,C 90.000,E1 115.207} C_DIS
LIN {X -0.084,Y -559.531,Z 753.435,A 0.000,B 0.000,C 90.000,E1 114.387} C_DIS
LIN {X -0.196,Y -560.883,Z 753.431,A 0.000,B 0.000,C 90.000,E1 113.567} C_DIS
LIN {X -0.199,Y -562.516,Z 753.425,A 0.000,B 0.000,C 90.000,E1 112.461} C_DIS
LIN {X 0.153,Y -564.386,Z 753.417,A 0.000,B 0.000,C 90.000,E1 111.046} C_DIS
LIN {X 0.004,Y -566.170,Z 753.409,A 0.000,B 0.000,C 90.000,E1 109.685} C_DIS
LIN {X 0.038,Y -567.784,Z 753.402,A 0.000,B 0.000,C 90.000,E1 108.308} C_DIS
LIN {X -0.051,Y -568.919,Z 753.396,A 0.000,B 0.000,C 90.000,E1 107.221} C_DIS
LIN {X -0.134,Y -570.090,Z 753.390,A 0.000,B 0.000,C 90.000,E1 106.134} C_DIS
LIN {X -0.182,Y -571.511,Z 753.382,A 0.000,B 0.000,C 90.000,E1 104.773} C_DIS
LIN {X 0.188,Y -573.454,Z 753.371,A 0.000,B 0.000,C 90.000,E1 102.827} C_DIS
LIN {X -0.083,Y -575.467,Z 753.361,A 0.000,B 0.000,C 90.000,E1 100.950} C_DIS
LIN {X -0.068,Y -577.115,Z 753.352,A 0.000,B 0.000,C 90.000,E1 99.321} C_DIS
LIN {X -0.094,Y -577.877,Z 753.347,A 0.000,B 0.000,C 90.000,E1 98.511} C_DIS
LIN {X -0.120,Y -579.256,Z 753.338,A 0.000,B 0.000,C 90.000,E1 96.891} C_DIS
LIN {X 0.022,Y -580.226,Z 753.332,A 0.000,B 0.000,C 90.000,E1 95.796} C_DIS
LIN {X -0.241,Y -581.229,Z 753.325,A 0.000,B 0.000,C 90.000,E1 94.473} C_DIS
LIN {X -0.116,Y -581.975,Z 753.319,A 0.000,B 0.000,C 90.000,E1 93.383} C_DIS
LIN {X 0.200,Y -582.871,Z 753.311,A 0.000,B 0.000,C 90.000,E1 92.007} C_DIS
LIN {X -0.236,Y -583.557,Z 753.305,A 0.000,B 0.000,C 90.000,E1 90.974} C_DIS
LIN {X 0.090,Y -584.256,Z 753.298,A 0.000,B 0.000,C 90.000,E1 89.599} C_DIS
LIN {X 0.041,Y -584.851,Z 753.289,A 0.000,B 0.000,C 90.000,E1 87.993} C_DIS
LIN {X 0.005,Y -585.384,Z 753.280,A 0.000,B 0.000,C 90.000,E1 86.388} C_DIS
LIN {X -0.171,Y -585.636,Z 753.273,A 0.000,B 0.000,C 90.000,E1 85.065} C_DIS
LIN {X 0.066,Y -585.824,Z 753.267,A 0.000,B 0.000,C 90.000,E1 83.970} C_DIS
LIN {X -0.109,Y -585.939,Z 753.259,A 0.000,B 0.000,C 90.000,E1 82.648} C_DIS
LIN {X 0.026,Y -585.970,Z 753.250,A 0.000,B 0.000,C 90.000,E1 81.027} C_DIS
LIN {X 0.006,Y -585.817,Z 753.243,A 0.000,B 0.000,C 90.000,E1 79.690} C_DIS
LIN {X -0.228,Y -585.433,Z 753.234,A 0.000,B 0.000,C 90.000,E1 78.105} C_DIS
LIN {X 0.189,Y -585.105,Z 753.228,A 0.000,B 0.000,C 90.000,E1 76.992} C_DIS
LIN {X -0.064,Y -584.472,Z 753.219,A 0.000,B 0.000,C 90.000,E1 75.408} C_DIS
LIN {X 0.133,Y -583.802,Z 753.211,A 0.000,B 0.000,C 90.000,E1 74.047} C_DIS
LIN {X 0.254,Y -583.257,Z 753.206,A 0.000,B 0.000,C 90.000,E1 72.960} C_DIS
LIN {X 0.039,Y -582.390,Z 753.198,A 0.000,B 0.000,C 90.000,E1 71.638} C_DIS
LIN {X 0.147,Y -581.640,Z 753.192,A 0.000,B 0.000,C 90.000,E1 70.550} C_DIS
LIN {X -0.059,Y -580.393,Z 753.183,A 0.000,B 0.000,C 90.000,E1 68.954} C_DIS
LIN {X -0.293,Y -578.861,Z 753.174,A 0.000,B 0.000,C 90.000,E1 67.358} C_DIS
LIN {X 0.184,Y -577.710,Z 753.168,A 0.000,B 0.000,C 90.000,E1 66.230} C_DIS
LIN {X -0.271,Y -576.052,Z 753.161,A 0.000,B 0.000,C 90.000,E1 64.921} C_DIS
LIN {X -0.109,Y -574.539,Z 753.155,A 0.000,B 0.000,C 90.000,E1 63.819} C_DIS
LIN {X -0.061,Y -573.223,Z 753.150,A 0.000,B 0.000,C 90.000,E1 62.999} C_DIS
LIN {X 0.068,Y -571.348,Z 753.144,A 0.000,B 0.000,C 90.000,E1 61.897} C_DIS
LIN {X 0.167,Y -569.092,Z 753.138,A 0.000,B 0.000,C 90.000,E1 60.795} C_DIS
LIN {X -0.084,Y -567.223,Z 753.133,A 0.000,B 0.000,C 90.000,E1 59.999} C_DIS
LIN {X 0.234,Y -564.423,Z 753.127,A 0.000,B 0.000,C 90.000,E1 58.869} C_DIS
LIN {X -0.066,Y -562.105,Z 753.123,A 0.000,B 0.000,C 90.000,E1 58.074} C_DIS
LIN {X -0.092,Y -559.566,Z 753.118,A 0.000,B 0.000,C 90.000,E1 57.248} C_DIS
LIN {X -0.140,Y -556.743,Z 753.113,A 0.000,B 0.000,C 90.000,E1 56.421} C_DIS
LIN {X -0.217,Y -553.698,Z 753.109,A 0.000,B 0.000,C 90.000,E1 55.595} C_DIS
LIN {X -0.076,Y -551.536,Z 753.106,A 0.000,B 0.000,C 90.000,E1 55.022} C_DIS
LIN {X -0.210,Y -547.864,Z 753.101,A 0.000,B 0.000,C 90.000,E1 54.196} C_DIS
LIN {X -0.252,Y -544.467,Z 753.097,A 0.000,B 0.000,C 90.000,E1 53.497} C_DIS
LIN {X -0.002,Y -540.738,Z 753.093,A 0.000,B 0.000,C 90.000,E1 52.763} C_DIS
LIN {X 0.043,Y -537.591,Z 753.090,A 0.000,B 0.000,C 90.000,E1 52.190} C_DIS
LIN {X 0.061,Y -534.158,Z 753.087,A 0.000,B 0.000,C 90.000,E1 51.618} C_DIS
LIN {X 0.054,Y -530.270,Z 753.084,A 0.000,B 0.000,C 90.000,E1 51.045} C_DIS
LIN {X -0.058,Y -525.988,Z 753.080,A 0.000,B 0.000,C 90.000,E1 50.481} C_DIS
LIN {X -0.125,Y -521.234,Z 753.077,A 0.000,B 0.000,C 90.000,E1 49.908} C_DIS
LIN {X 0.202,Y -515.875,Z 753.074,A 0.000,B 0.000,C 90.000,E1 49.299} C_DIS
LIN {X -0.248,Y -511.729,Z 753.072,A 0.000,B 0.000,C 90.000,E1 48.933} C_DIS
LIN {X -0.198,Y -505.812,Z 753.069,A 0.000,B 0.000,C 90.000,E1 48.405} C_DIS
LIN {X 0.075,Y -499.731,Z 753.066,A 0.000,B 0.000,C 90.000,E1 47.877} C_DIS
LIN {X -0.258,Y -495.110,Z 753.064,A 0.000,B 0.000,C 90.000,E1 47.553} C_DIS
LIN {X -0.092,Y -483.891,Z 753.060,A 0.000,B 0.000,C 90.000,E1 46.743} C_DIS
LIN {X 0.287,Y -467.588,Z 753.054,A 0.000,B 0.000,C 90.000,E1 45.648} C_DIS
LIN {X 0.048,Y -449.734,Z 753.047,A 0.000,B 0.000,C 90.000,E1 44.514} C_DIS
LIN {X 0.020,Y -425.570,Z 753.038,A 0.000,B 0.000,C 90.000,E1 42.852} C_DIS
LIN {X -0.042,Y -416.519,Z 753.034,A 0.000,B 0.000,C 90.000,E1 42.162} C_DIS
LIN {X -0.109,Y -411.704,Z 753.032,A 0.000,B 0.000,C 90.000,E1 41.757} C_DIS
LIN {X -0.139,Y -411.693,Z 753.032,A 0.000,B 0.000,C 90.000,E1 41.757} C_DIS
LIN {X 0.073,Y -405.661,Z 753.013,A 0.000,B 0.000,C 90.000,E1 38.382} C_DIS
LIN {X 0.061,Y -401.224,Z 753.002,A 0.000,B 0.000,C 90.000,E1 36.297} C_DIS
LIN {X -0.041,Y -401.034,Z 753.001,A 0.000,B 0.000,C 90.000,E1 36.137} C_DIS
LIN {X -0.051,Y -401.498,Z 752.984,A 0.000,B 0.000,C 90.000,E1 33.166} C_DIS
LIN {X 0.066,Y -402.226,Z 752.973,A 0.000,B 0.000,C 90.000,E1 31.052} C_DIS
LIN {X 0.028,Y -403.418,Z 752.959,A 0.000,B 0.000,C 90.000,E1 28.615} C_DIS
LIN {X 0.006,Y -404.738,Z 752.945,A 0.000,B 0.000,C 90.000,E1 26.181} C_DIS
LIN {X 0.112,Y -406.718,Z 752.930,A 0.000,B 0.000,C 90.000,E1 23.387} C_DIS
LIN {X -0.114,Y -410.583,Z 752.907,A 0.000,B 0.000,C 90.000,E1 19.268} C_DIS
LIN {X 0.043,Y -413.993,Z 752.892,A 0.000,B 0.000,C 90.000,E1 16.496} C_DIS
LIN {X -0.228,Y -416.898,Z 752.880,A 0.000,B 0.000,C 90.000,E1 14.481} C_DIS
LIN {X 0.034,Y -420.573,Z 752.867,A 0.000,B 0.000,C 90.000,E1 12.063} C_DIS
LIN {X 0.061,Y -423.316,Z 752.858,A 0.000,B 0.000,C 90.000,E1 10.366} C_DIS
LIN {X 0.089,Y -426.550,Z 752.846,A 0.000,B 0.000,C 90.000,E1 8.341} C_DIS
LIN {X 0.200,Y -429.798,Z 752.835,A 0.000,B 0.000,C 90.000,E1 6.315} C_DIS
LIN {X 0.051,Y -434.393,Z 752.820,A 0.000,B 0.000,C 90.000,E1 3.669} C_DIS
LIN {X 0.103,Y -437.441,Z 752.811,A 0.000,B 0.000,C 90.000,E1 2.007} C_DIS
LIN {X 0.000,Y -441.274,Z 752.800,A 0.000,B 0.000,C 90.000,E1 360.000} C_DIS
LIN {X -0.220,Y -444.264,Z 752.792,A 0.000,B 0.000,C 90.000,E1 358.511} C_DIS
LIN {X 0.190,Y -448.439,Z 752.781,A 0.000,B 0.000,C 90.000,E1 356.502} C_DIS
LIN {X -0.092,Y -454.961,Z 752.765,A 0.000,B 0.000,C 90.000,E1 353.628} C_DIS
LIN {X 0.039,Y -458.613,Z 752.756,A 0.000,B 0.000,C 90.000,E1 352.008} C_DIS
LIN {X -0.211,Y -462.061,Z 752.747,A 0.000,B 0.000,C 90.000,E1 350.443} C_DIS
LIN {X 0.080,Y -464.023,Z 752.742,A 0.000,B 0.000,C 90.000,E1 349.454} C_DIS
LIN {X 0.003,Y -467.103,Z 752.733,A 0.000,B 0.000,C 90.000,E1 347.881} C_DIS
LIN {X 0.097,Y -471.847,Z 752.719,A 0.000,B 0.000,C 90.000,E1 345.353} C_DIS
LIN {X -0.141,Y -473.179,Z 752.715,A 0.000,B 0.000,C 90.000,E1 344.755} C_DIS
LIN {X 0.263,Y -473.954,Z 752.714,A 0.000,B 0.000,C 90.000,E1 344.393} C_DIS
LIN {X 0.046,Y -475.831,Z 752.710,A 0.000,B 0.000,C 90.000,E1 343.795} C_DIS
LIN {X 0.086,Y -477.596,Z 752.707,A 0.000,B 0.000,C 90.000,E1 343.323} C_DIS
LIN {X 0.133,Y -479.962,Z 752.705,A 0.000,B 0.000,C 90.000,E1 342.851} C_DIS
LIN {X -0.046,Y -482.394,Z 752.703,A 0.000,B 0.000,C 90.000,E1 342.489} C_DIS
LIN {X -0.059,Y -485.278,Z 752.701,A 0.000,B 0.000,C 90.000,E1 342.127} C_DIS
LIN {X -0.184,Y -489.567,Z 752.698,A 0.000,B 0.000,C 90.000,E1 341.692} C_DIS
LIN {X 0.077,Y -493.418,Z 752.696,A 0.000,B 0.000,C 90.000,E1 341.329} C_DIS
LIN {X 0.004,Y -505.981,Z 752.691,A 0.000,B 0.000,C 90.000,E1 340.423} C_DIS
LIN {X 0.187,Y -518.619,Z 752.687,A 0.000,B 0.000,C 90.000,E1 339.571} C_DIS
LIN {X -0.162,Y -536.419,Z 752.681,A 0.000,B 0.000,C 90.000,E1 338.539} C_DIS
LIN {X 0.246,Y -542.479,Z 752.679,A 0.000,B 0.000,C 90.000,E1 338.103} C_DIS
LIN {X -0.070,Y -551.434,Z 752.675,A 0.000,B 0.000,C 90.000,E1 337.486} C_DIS
LIN {X 0.140,Y -556.887,Z 752.672,A 0.000,B 0.000,C 90.000,E1 336.997} C_DIS
LIN {X 0.249,Y -562.148,Z 752.670,A 0.000,B 0.000,C 90.000,E1 336.485} C_DIS
LIN {X -0.043,Y -568.278,Z 752.666,A 0.000,B 0.000,C 90.000,E1 335.869} C_DIS
LIN {X 0.164,Y -573.153,Z 752.663,A 0.000,B 0.000,C 90.000,E1 335.305} C_DIS
LIN {X -0.211,Y -578.928,Z 752.659,A 0.000,B 0.000,C 90.000,E1 334.665} C_DIS
LIN {X -0.143,Y -586.573,Z 752.654,A 0.000,B 0.000,C 90.000,E1 333.717} C_DIS
LIN {X 0.206,Y -594.708,Z 752.648,A 0.000,B 0.000,C 90.000,E1 332.615} C_DIS
LIN {X -0.097,Y -601.428,Z 752.643,A 0.000,B 0.000,C 90.000,E1 331.719} C_DIS
LIN {X -0.039,Y -607.882,Z 752.638,A 0.000,B 0.000,C 90.000,E1 330.795} C_DIS
LIN {X 0.121,Y -613.206,Z 752.633,A 0.000,B 0.000,C 90.000,E1 329.999} C_DIS
LIN {X -0.204,Y -619.081,Z 752.628,A 0.000,B 0.000,C 90.000,E1 329.125} C_DIS
LIN {X 0.062,Y -626.139,Z 752.622,A 0.000,B 0.000,C 90.000,E1 327.946} C_DIS
LIN {X -0.133,Y -629.128,Z 752.619,A 0.000,B 0.000,C 90.000,E1 327.454} C_DIS
LIN {X 0.066,Y -634.100,Z 752.614,A 0.000,B 0.000,C 90.000,E1 326.548} C_DIS
LIN {X 0.361,Y -639.951,Z 752.608,A 0.000,B 0.000,C 90.000,E1 325.388} C_DIS
LIN {X 0.190,Y -644.871,Z 752.602,A 0.000,B 0.000,C 90.000,E1 324.402} C_DIS
LIN {X 0.075,Y -649.538,Z 752.597,A 0.000,B 0.000,C 90.000,E1 323.417} C_DIS
LIN {X 0.009,Y -653.787,Z 752.591,A 0.000,B 0.000,C 90.000,E1 322.431} C_DIS
LIN {X -0.065,Y -656.878,Z 752.587,A 0.000,B 0.000,C 90.000,E1 321.698} C_DIS
LIN {X 0.328,Y -661.604,Z 752.580,A 0.000,B 0.000,C 90.000,E1 320.436} C_DIS
LIN {X 0.311,Y -665.143,Z 752.575,A 0.000,B 0.000,C 90.000,E1 319.461} C_DIS
LIN {X 0.338,Y -669.209,Z 752.568,A 0.000,B 0.000,C 90.000,E1 318.243} C_DIS
LIN {X -0.067,Y -672.960,Z 752.562,A 0.000,B 0.000,C 90.000,E1 317.067} C_DIS
LIN {X -0.444,Y -675.785,Z 752.556,A 0.000,B 0.000,C 90.000,E1 316.134} C_DIS
LIN {X -0.318,Y -678.348,Z 752.551,A 0.000,B 0.000,C 90.000,E1 315.162} C_DIS
LIN {X -0.157,Y -680.678,Z 752.545,A 0.000,B 0.000,C 90.000,E1 314.190} C_DIS
LIN {X 0.079,Y -683.394,Z 752.539,A 0.000,B 0.000,C 90.000,E1 312.975} C_DIS
LIN {X 0.336,Y -685.412,Z 752.534,A 0.000,B 0.000,C 90.000,E1 312.000} C_DIS
LIN {X -0.216,Y -688.108,Z 752.526,A 0.000,B 0.000,C 90.000,E1 310.620} C_DIS
LIN {X 0.113,Y -689.577,Z 752.520,A 0.000,B 0.000,C 90.000,E1 309.644} C_DIS
LIN {X -0.140,Y -690.579,Z 752.516,A 0.000,B 0.000,C 90.000,E1 308.955} C_DIS
LIN {X 0.022,Y -692.347,Z 752.509,A 0.000,B 0.000,C 90.000,E1 307.523} C_DIS
LIN {X -0.028,Y -693.382,Z 752.503,A 0.000,B 0.000,C 90.000,E1 306.583} C_DIS
LIN {X -0.212,Y -694.641,Z 752.495,A 0.000,B 0.000,C 90.000,E1 305.185} C_DIS
LIN {X -0.022,Y -695.635,Z 752.489,A 0.000,B 0.000,C 90.000,E1 303.992} C_DIS
LIN {X 0.411,Y -696.719,Z 752.481,A 0.000,B 0.000,C 90.000,E1 302.546} C_DIS
LIN {X 0.142,Y -697.952,Z 752.472,A 0.000,B 0.000,C 90.000,E1 300.924} C_DIS
LIN {X -0.292,Y -698.372,Z 752.468,A 0.000,B 0.000,C 90.000,E1 300.256} C_DIS
LIN {X -0.202,Y -698.797,Z 752.461,A 0.000,B 0.000,C 90.000,E1 299.077} C_DIS
LIN {X -0.190,Y -699.313,Z 752.452,A 0.000,B 0.000,C 90.000,E1 297.436} C_DIS
LIN {X -0.272,Y -700.298,Z 752.441,A 0.000,B 0.000,C 90.000,E1 295.335} C_DIS
LIN {X 0.247,Y -700.380,Z 752.437,A 0.000,B 0.000,C 90.000,E1 294.591} C_DIS
LIN {X 0.149,Y -699.711,Z 752.434,A 0.000,B 0.000,C 90.000,E1 294.131} C_DIS
LIN {X 0.132,Y -699.125,Z 752.433,A 0.000,B 0.000,C 90.000,E1 293.898} C_DIS
LIN {X -0.256,Y -696.614,Z 752.430,A 0.000,B 0.000,C 90.000,E1 293.462} C_DIS
LIN {X -0.127,Y -695.912,Z 752.430,A 0.000,B 0.000,C 90.000,E1 293.334} C_DIS
LIN {X 0.001,Y -694.896,Z 752.429,A 0.000,B 0.000,C 90.000,E1 293.206} C_DIS
LIN {X 0.126,Y -693.368,Z 752.428,A 0.000,B 0.000,C 90.000,E1 293.078} C_DIS
LIN {X -0.226,Y -689.861,Z 752.427,A 0.000,B 0.000,C 90.000,E1 292.898} C_DIS
LIN {X 0.121,Y -686.554,Z 752.426,A 0.000,B 0.000,C 90.000,E1 292.695} C_DIS
LIN {X -0.223,Y -684.437,Z 752.426,A 0.000,B 0.000,C 90.000,E1 292.642} C_DIS
LIN {X 0.013,Y -676.083,Z 752.425,A 0.000,B 0.000,C 90.000,E1 292.408} C_DIS
LIN {X 0.138,Y -668.452,Z 752.424,A 0.000,B 0.000,C 90.000,E1 292.280} C_DIS
LIN {X -0.224,Y -655.405,Z 752.423,A 0.000,B 0.000,C 90.000,E1 292.153} C_DIS
LIN {X 0.057,Y -645.303,Z 752.422,A 0.000,B 0.000,C 90.000,E1 291.972} C_DIS
LIN {X -0.059,Y -632.226,Z 752.421,A 0.000,B 0.000,C 90.000,E1 291.716} C_DIS
LIN {X -0.160,Y -611.711,Z 752.418,A 0.000,B 0.000,C 90.000,E1 291.227} C_DIS
LIN {X 0.041,Y -575.092,Z 752.412,A 0.000,B 0.000,C 90.000,E1 290.174} C_DIS
LIN {X -0.042,Y -566.130,Z 752.411,A 0.000,B 0.000,C 90.000,E1 289.939} C_DIS
LIN {X -0.177,Y -560.944,Z 752.410,A 0.000,B 0.000,C 90.000,E1 289.758} C_DIS
LIN {X -0.227,Y -557.416,Z 752.409,A 0.000,B 0.000,C 90.000,E1 289.577} C_DIS
LIN {X -0.132,Y -555.896,Z 752.408,A 0.000,B 0.000,C 90.000,E1 289.396} C_DIS
LIN {X -0.161,Y -555.880,Z 752.408,A 0.000,B 0.000,C 90.000,E1 289.396} C_DIS
LIN {X -0.003,Y -555.213,Z 752.406,A 0.000,B 0.000,C 90.000,E1 289.087} C_DIS
LIN {X 0.207,Y -554.767,Z 752.403,A 0.000,B 0.000,C 90.000,E1 288.489} C_DIS
LIN {X -0.175,Y -554.551,Z 752.398,A 0.000,B 0.000,C 90.000,E1 287.692} C_DIS
LIN {X -0.232,Y -553.908,Z 752.389,A 0.000,B 0.000,C 90.000,E1 286.024} C_DIS
LIN {X -0.181,Y -553.199,Z 752.378,A 0.000,B 0.000,C 90.000,E1 284.064} C_DIS
LIN {X 0.129,Y -552.607,Z 752.369,A 0.000,B 0.000,C 90.000,E1 282.355} C_DIS
LIN {X 0.305,Y -552.108,Z 752.359,A 0.000,B 0.000,C 90.000,E1 280.658} C_DIS
LIN {X 0.250,Y -551.519,Z 752.352,A 0.000,B 0.000,C 90.000,E1 279.265} C_DIS
LIN {X 0.073,Y -551.043,Z 752.345,A 0.000,B 0.000,C 90.000,E1 278.163} C_DIS
LIN {X -0.078,Y -550.434,Z 752.338,A 0.000,B 0.000,C 90.000,E1 276.777} C_DIS
LIN {X 0.165,Y -550.054,Z 752.333,A 0.000,B 0.000,C 90.000,E1 275.910} C_DIS
LIN {X -0.063,Y -549.214,Z 752.325,A 0.000,B 0.000,C 90.000,E1 274.531} C_DIS
LIN {X -0.216,Y -548.127,Z 752.314,A 0.000,B 0.000,C 90.000,E1 272.579} C_DIS
LIN {X 0.084,Y -547.220,Z 752.305,A 0.000,B 0.000,C 90.000,E1 270.859} C_DIS
LIN {X -0.238,Y -546.367,Z 752.297,A 0.000,B 0.000,C 90.000,E1 269.484} C_DIS
LIN {X 0.023,Y -545.209,Z 752.288,A 0.000,B 0.000,C 90.000,E1 267.764} C_DIS
LIN {X 0.253,Y -544.174,Z 752.278,A 0.000,B 0.000,C 90.000,E1 266.045} C_DIS
LIN {X -0.079,Y -543.255,Z 752.270,A 0.000,B 0.000,C 90.000,E1 264.666} C_DIS
LIN {X 0.169,Y -542.251,Z 752.263,A 0.000,B 0.000,C 90.000,E1 263.223} C_DIS
LIN {X -0.214,Y -541.600,Z 752.258,A 0.000,B 0.000,C 90.000,E1 262.413} C_DIS
LIN {X 0.073,Y -540.162,Z 752.248,A 0.000,B 0.000,C 90.000,E1 260.679} C_DIS
LIN {X -0.167,Y -539.215,Z 752.242,A 0.000,B 0.000,C 90.000,E1 259.567} C_DIS
LIN {X 0.075,Y -538.077,Z 752.234,A 0.000,B 0.000,C 90.000,E1 258.117} C_DIS
LIN {X -0.076,Y -537.078,Z 752.228,A 0.000,B 0.000,C 90.000,E1 256.992} C_DIS
LIN {X 0.161,Y -536.062,Z 752.221,A 0.000,B 0.000,C 90.000,E1 255.825} C_DIS
LIN {X -0.014,Y -534.821,Z 752.215,A 0.000,B 0.000,C 90.000,E1 254.700} C_DIS
LIN {X -0.060,Y -533.549,Z 752.209,A 0.000,B 0.000,C 90.000,E1 253.559} C_DIS
LIN {X 0.102,Y -531.629,Z 752.199,A 0.000,B 0.000,C 90.000,E1 251.819} C_DIS
LIN {X 0.000,Y -530.691,Z 752.194,A 0.000,B 0.000,C 90.000,E1 250.967} C_DIS
LIN {X -0.236,Y -528.329,Z 752.185,A 0.000,B 0.000,C 90.000,E1 249.263} C_DIS
LIN {X -0.024,Y -526.289,Z 752.177,A 0.000,B 0.000,C 90.000,E1 247.794} C_DIS
LIN {X 0.023,Y -523.667,Z 752.167,A 0.000,B 0.000,C 90.000,E1 246.049} C_DIS
LIN {X -0.077,Y -521.822,Z 752.161,A 0.000,B 0.000,C 90.000,E1 244.897} C_DIS
LIN {X 0.045,Y -519.893,Z 752.154,A 0.000,B 0.000,C 90.000,E1 243.717} C_DIS
LIN {X -0.241,Y -518.379,Z 752.149,A 0.000,B 0.000,C 90.000,E1 242.871} C_DIS
LIN {X -0.055,Y -515.674,Z 752.141,A 0.000,B 0.000,C 90.000,E1 241.385} C_DIS
LIN {X -0.029,Y -512.248,Z 752.131,A 0.000,B 0.000,C 90.000,E1 239.616} C_DIS
LIN {X -0.261,Y -508.811,Z 752.121,A 0.000,B 0.000,C 90.000,E1 237.867} C_DIS
LIN {X 0.194,Y -506.319,Z 752.115,A 0.000,B 0.000,C 90.000,E1 236.628} C_DIS
LIN {X 0.017,Y -504.333,Z 752.110,A 0.000,B 0.000,C 90.000,E1 235.754} C_DIS
LIN {X -0.132,Y -500.853,Z 752.102,A 0.000,B 0.000,C 90.000,E1 234.276} C_DIS
LIN {X 0.082,Y -497.903,Z 752.095,A 0.000,B 0.000,C 90.000,E1 233.050} C_DIS
LIN {X 0.084,Y -495.624,Z 752.090,A 0.000,B 0.000,C 90.000,E1 232.145} C_DIS
LIN {X -0.158,Y -489.612,Z 752.076,A 0.000,B 0.000,C 90.000,E1 229.747} C_DIS
LIN {X -0.059,Y -484.781,Z 752.064,A 0.000,B 0.000,C 90.000,E1 227.595} C_DIS
LIN {X -0.023,Y -481.492,Z 752.056,A 0.000,B 0.000,C 90.000,E1 226.053} C_DIS
LIN {X 0.049,Y -477.572,Z 752.046,A 0.000,B 0.000,C 90.000,E1 224.190} C_DIS
LIN {X 0.270,Y -474.242,Z 752.037,A 0.000,B 0.000,C 90.000,E1 222.609} C_DIS
LIN {X 0.241,Y -472.283,Z 752.032,A 0.000,B 0.000,C 90.000,E1 221.676} C_DIS
LIN {X 0.225,Y -467.377,Z 752.020,A 0.000,B 0.000,C 90.000,E1 219.483} C_DIS
LIN {X 0.102,Y -463.294,Z 752.009,A 0.000,B 0.000,C 90.000,E1 217.604} C_DIS
LIN {X 0.005,Y -458.666,Z 751.997,A 0.000,B 0.000,C 90.000,E1 215.391} C_DIS
LIN {X 0.063,Y -455.422,Z 751.988,A 0.000,B 0.000,C 90.000,E1 213.785} C_DIS
LIN {X -0.101,Y -451.689,Z 751.977,A 0.000,B 0.000,C 90.000,E1 211.878} C_DIS
LIN {X 0.025,Y -448.055,Z 751.966,A 0.000,B 0.000,C 90.000,E1 209.922} C_DIS
LIN {X 0.092,Y -445.618,Z 751.959,A 0.000,B 0.000,C 90.000,E1 208.615} C_DIS
LIN {X -0.085,Y -443.287,Z 751.952,A 0.000,B 0.000,C 90.000,E1 207.334} C_DIS
LIN {X 0.178,Y -439.528,Z 751.941,A 0.000,B 0.000,C 90.000,E1 205.335} C_DIS
LIN {X 0.134,Y -436.449,Z 751.932,A 0.000,B 0.000,C 90.000,E1 203.695} C_DIS
LIN {X -0.146,Y -433.369,Z 751.923,A 0.000,B 0.000,C 90.000,E1 202.078} C_DIS
LIN {X 0.127,Y -431.543,Z 751.917,A 0.000,B 0.000,C 90.000,E1 201.046} C_DIS
LIN {X 0.013,Y -427.100,Z 751.904,A 0.000,B 0.000,C 90.000,E1 198.725} C_DIS
LIN {X -0.153,Y -423.222,Z 751.893,A 0.000,B 0.000,C 90.000,E1 196.732} C_DIS
LIN {X -0.084,Y -418.615,Z 751.880,A 0.000,B 0.000,C 90.000,E1 194.356} C_DIS
LIN {X 0.021,Y -414.906,Z 751.868,A 0.000,B 0.000,C 90.000,E1 192.299} C_DIS
LIN {X -0.048,Y -411.376,Z 751.857,A 0.000,B 0.000,C 90.000,E1 190.254} C_DIS
LIN {X 0.080,Y -409.046,Z 751.849,A 0.000,B 0.000,C 90.000,E1 188.859} C_DIS
LIN {X 0.145,Y -405.034,Z 751.836,A 0.000,B 0.000,C 90.000,E1 186.429} C_DIS
LIN {X -0.046,Y -400.812,Z 751.820,A 0.000,B 0.000,C 90.000,E1 183.669} C_DIS
LIN {X -0.189,Y -395.688,Z 751.799,A 0.000,B 0.000,C 90.000,E1 179.828} C_DIS
LIN {X 0.064,Y -392.616,Z 751.783,A 0.000,B 0.000,C 90.000,E1 176.963} C_DIS
LIN {X -0.172,Y -389.620,Z 751.765,A 0.000,B 0.000,C 90.000,E1 173.799} C_DIS
LIN {X -0.094,Y -387.373,Z 751.744,A 0.000,B 0.000,C 90.000,E1 169.859} C_DIS
LIN {X -0.099,Y -386.154,Z 751.730,A 0.000,B 0.000,C 90.000,E1 167.353} C_DIS
LIN {X 0.173,Y -385.370,Z 751.720,A 0.000,B 0.000,C 90.000,E1 165.519} C_DIS
LIN {X 0.097,Y -384.571,Z 751.706,A 0.000,B 0.000,C 90.000,E1 163.015} C_DIS
LIN {X -0.101,Y -383.756,Z 751.688,A 0.000,B 0.000,C 90.000,E1 159.806} C_DIS
LIN {X -0.089,Y -383.383,Z 751.674,A 0.000,B 0.000,C 90.000,E1 157.283} C_DIS
LIN {X 0.205,Y -383.257,Z 751.660,A 0.000,B 0.000,C 90.000,E1 154.717} C_DIS
LIN {X -0.075,Y -385.429,Z 751.628,A 0.000,B 0.000,C 90.000,E1 148.997} C_DIS
LIN {X -0.078,Y -389.013,Z 751.606,A 0.000,B 0.000,C 90.000,E1 145.055} C_DIS
LIN {X -0.131,Y -392.071,Z 751.594,A 0.000,B 0.000,C 90.000,E1 142.924} C_DIS
LIN {X 0.110,Y -394.161,Z 751.588,A 0.000,B 0.000,C 90.000,E1 141.823} C_DIS
LIN {X 0.040,Y -395.846,Z 751.584,A 0.000,B 0.000,C 90.000,E1 141.126} C_DIS
LIN {X -0.080,Y -398.585,Z 751.579,A 0.000,B 0.000,C 90.000,E1 140.275} C_DIS
LIN {X -0.074,Y -400.839,Z 751.576,A 0.000,B 0.000,C 90.000,E1 139.747} C_DIS
LIN {X 0.163,Y -404.600,Z 751.572,A 0.000,B 0.000,C 90.000,E1 139.013} C_DIS
LIN {X -0.008,Y -408.559,Z 751.569,A 0.000,B 0.000,C 90.000,E1 138.485} C_DIS
LIN {X 0.004,Y -413.275,Z 751.566,A 0.000,B 0.000,C 90.000,E1 137.919} C_DIS
LIN {X 0.058,Y -422.901,Z 751.561,A 0.000,B 0.000,C 90.000,E1 136.905} C_DIS
LIN {X -0.132,Y -431.790,Z 751.556,A 0.000,B 0.000,C 90.000,E1 136.053} C_DIS
LIN {X -0.063,Y -443.296,Z 751.549,A 0.000,B 0.000,C 90.000,E1 134.879} C_DIS
LIN {X -0.247,Y -451.923,Z 751.544,A 0.000,B 0.000,C 90.000,E1 134.028} C_DIS
LIN {X 0.078,Y -458.902,Z 751.540,A 0.000,B 0.000,C 90.000,E1 133.257} C_DIS
LIN {X 0.095,Y -467.214,Z 751.535,A 0.000,B 0.000,C 90.000,E1 132.366} C_DIS
LIN {X 0.320,Y -472.511,Z 751.532,A 0.000,B 0.000,C 90.000,E1 131.757} C_DIS
LIN {X -0.163,Y -479.275,Z 751.528,A 0.000,B 0.000,C 90.000,E1 131.067} C_DIS
LIN {X 0.076,Y -487.953,Z 751.522,A 0.000,B 0.000,C 90.000,E1 130.011} C_DIS
LIN {X 0.086,Y -492.888,Z 751.519,A 0.000,B 0.000,C 90.000,E1 129.402} C_DIS
LIN {X 0.007,Y -497.391,Z 751.516,A 0.000,B 0.000,C 90.000,E1 128.830} C_DIS
LIN {X 0.056,Y -501.695,Z 751.512,A 0.000,B 0.000,C 90.000,E1 128.222} C_DIS
LIN {X 0.084,Y -505.639,Z 751.509,A 0.000,B 0.000,C 90.000,E1 127.649} C_DIS
LIN {X -0.001,Y -510.428,Z 751.505,A 0.000,B 0.000,C 90.000,E1 126.916} C_DIS
LIN {X 0.235,Y -514.043,Z 751.502,A 0.000,B 0.000,C 90.000,E1 126.297} C_DIS
LIN {X 0.021,Y -519.217,Z 751.497,A 0.000,B 0.000,C 90.000,E1 125.438} C_DIS
LIN {X -0.040,Y -520.909,Z 751.495,A 0.000,B 0.000,C 90.000,E1 125.152} C_DIS
LIN {X 0.034,Y -527.408,Z 751.488,A 0.000,B 0.000,C 90.000,E1 123.833} C_DIS
LIN {X -0.076,Y -533.205,Z 751.481,A 0.000,B 0.000,C 90.000,E1 122.546} C_DIS
LIN {X -0.087,Y -537.494,Z 751.475,A 0.000,B 0.000,C 90.000,E1 121.544} C_DIS
LIN {X 0.090,Y -540.912,Z 751.470,A 0.000,B 0.000,C 90.000,E1 120.669} C_DIS
LIN {X 0.300,Y -544.074,Z 751.466,A 0.000,B 0.000,C 90.000,E1 119.795} C_DIS
LIN {X 0.275,Y -547.055,Z 751.461,A 0.000,B 0.000,C 90.000,E1 118.949} C_DIS
LIN {X -0.200,Y -549.890,Z 751.456,A 0.000,B 0.000,C 90.000,E1 118.153} C_DIS
LIN {X -0.167,Y -552.607,Z 751.452,A 0.000,B 0.000,C 90.000,E1 117.308} C_DIS
LIN {X 0.141,Y -555.106,Z 751.447,A 0.000,B 0.000,C 90.000,E1 116.437} C_DIS
LIN {X 0.231,Y -557.170,Z 751.442,A 0.000,B 0.000,C 90.000,E1 115.591} C_DIS
LIN {X 0.098,Y -558.935,Z 751.438,A 0.000,B 0.000,C 90.000,E1 114.771} C_DIS
LIN {X -0.223,Y -560.810,Z 751.432,A 0.000,B 0.000,C 90.000,E1 113.695} C_DIS
LIN {X -0.228,Y -562.487,Z 751.425,A 0.000,B 0.000,C 90.000,E1 112.589} C_DIS
LIN {X -0.074,Y -564.758,Z 751.416,A 0.000,B 0.000,C 90.000,E1 110.918} C_DIS
LIN {X -0.018,Y -566.215,Z 751.410,A 0.000,B 0.000,C 90.000,E1 109.812} C_DIS
LIN {X -0.184,Y -568.176,Z 751.401,A 0.000,B 0.000,C 90.000,E1 108.181} C_DIS
LIN {X 0.104,Y -569.046,Z 751.396,A 0.000,B 0.000,C 90.000,E1 107.330} C_DIS
LIN {X -0.142,Y -570.257,Z 751.390,A 0.000,B 0.000,C 90.000,E1 106.260} C_DIS
LIN {X 0.152,Y -571.957,Z 751.381,A 0.000,B 0.000,C 90.000,E1 104.592} C_DIS
LIN {X -0.031,Y -573.943,Z 751.371,A 0.000,B 0.000,C 90.000,E1 102.703} C_DIS
LIN {X -0.052,Y -575.710,Z 751.362,A 0.000,B 0.000,C 90.000,E1 101.074} C_DIS
LIN {X -0.022,Y -577.353,Z 751.352,A 0.000,B 0.000,C 90.000,E1 99.443} C_DIS
LIN {X 0.175,Y -578.383,Z 751.346,A 0.000,B 0.000,C 90.000,E1 98.341} C_DIS
LIN {X -0.046,Y -580.330,Z 751.334,A 0.000,B 0.000,C 90.000,E1 96.201} C_DIS
LIN {X -0.305,Y -581.396,Z 751.327,A 0.000,B 0.000,C 90.000,E1 94.878} C_DIS
LIN {X 0.035,Y -582.341,Z 751.320,A 0.000,B 0.000,C 90.000,E1 93.498} C_DIS
LIN {X -0.048,Y -583.454,Z 751.311,A 0.000,B 0.000,C 90.000,E1 91.892} C_DIS
LIN {X -0.074,Y -583.970,Z 751.306,A 0.000,B 0.000,C 90.000,E1 91.088} C_DIS
LIN {X 0.258,Y -584.674,Z 751.299,A 0.000,B 0.000,C 90.000,E1 89.714} C_DIS
LIN {X 0.219,Y -585.298,Z 751.290,A 0.000,B 0.000,C 90.000,E1 88.108} C_DIS
LIN {X 0.194,Y -585.845,Z 751.281,A 0.000,B 0.000,C 90.000,E1 86.502} C_DIS
LIN {X -0.201,Y -586.067,Z 751.275,A 0.000,B 0.000,C 90.000,E1 85.469} C_DIS
LIN {X 0.214,Y -586.313,Z 751.267,A 0.000,B 0.000,C 90.000,E1 84.090} C_DIS
LIN {X -0.226,Y -586.426,Z 751.258,A 0.000,B 0.000,C 90.000,E1 82.527} C_DIS
LIN {X -0.070,Y -586.414,Z 751.250,A 0.000,B 0.000,C 90.000,E1 80.905} C_DIS
LIN {X -0.073,Y -586.227,Z 751.242,A 0.000,B 0.000,C 90.000,E1 79.567} C_DIS
LIN {X 0.162,Y -585.814,Z 751.233,A 0.000,B 0.000,C 90.000,E1 77.937} C_DIS
LIN {X -0.240,Y -585.568,Z 751.229,A 0.000,B 0.000,C 90.000,E1 77.173} C_DIS
LIN {X 0.227,Y -584.894,Z 751.220,A 0.000,B 0.000,C 90.000,E1 75.519} C_DIS
LIN {X -0.124,Y -584.222,Z 751.212,A 0.000,B 0.000,C 90.000,E1 74.212} C_DIS
LIN {X 0.067,Y -583.491,Z 751.205,A 0.000,B 0.000,C 90.000,E1 72.851} C_DIS
LIN {X -0.030,Y -582.972,Z 751.200,A 0.000,B 0.000,C 90.000,E1 72.054} C_DIS
LIN {X -0.251,Y -582.027,Z 751.193,A 0.000,B 0.000,C 90.000,E1 70.732} C_DIS
LIN {X 0.094,Y -580.737,Z 751.184,A 0.000,B 0.000,C 90.000,E1 69.082} C_DIS
LIN {X -0.135,Y -579.190,Z 751.175,A 0.000,B 0.000,C 90.000,E1 67.486} C_DIS
LIN {X -0.040,Y -578.334,Z 751.170,A 0.000,B 0.000,C 90.000,E1 66.666} C_DIS
LIN {X 0.044,Y -576.691,Z 751.163,A 0.000,B 0.000,C 90.000,E1 65.305} C_DIS
LIN {X -0.041,Y -575.230,Z 751.157,A 0.000,B 0.000,C 90.000,E1 64.229} C_DIS
LIN {X 0.265,Y -574.039,Z 751.152,A 0.000,B 0.000,C 90.000,E1 63.384} C_DIS
LIN {X 0.139,Y -572.103,Z 751.146,A 0.000,B 0.000,C 90.000,E1 62.308} C_DIS
LIN {X 0.078,Y -571.112,Z 751.143,A 0.000,B 0.000,C 90.000,E1 61.769} C_DIS
LIN {X 0.172,Y -568.714,Z 751.137,A 0.000,B 0.000,C 90.000,E1 60.667} C_DIS
LIN {X -0.083,Y -566.769,Z 751.133,A 0.000,B 0.000,C 90.000,E1 59.871} C_DIS
LIN {X 0.226,Y -563.884,Z 751.127,A 0.000,B 0.000,C 90.000,E1 58.742} C_DIS
LIN {X 0.217,Y -561.482,Z 751.122,A 0.000,B 0.000,C 90.000,E1 57.916} C_DIS
LIN {X -0.114,Y -558.843,Z 751.117,A 0.000,B 0.000,C 90.000,E1 57.120} C_DIS
LIN {X -0.094,Y -554.884,Z 751.111,A 0.000,B 0.000,C 90.000,E1 56.008} C_DIS
LIN {X -0.019,Y -553.905,Z 751.110,A 0.000,B 0.000,C 90.000,E1 55.722} C_DIS
LIN {X -0.126,Y -550.503,Z 751.105,A 0.000,B 0.000,C 90.000,E1 54.895} C_DIS
LIN {X -0.142,Y -547.365,Z 751.101,A 0.000,B 0.000,C 90.000,E1 54.196} C_DIS
LIN {X -0.188,Y -543.884,Z 751.097,A 0.000,B 0.000,C 90.000,E1 53.497} C_DIS
LIN {X -0.122,Y -540.918,Z 751.094,A 0.000,B 0.000,C 90.000,E1 52.924} C_DIS
LIN {X 0.094,Y -536.838,Z 751.090,A 0.000,B 0.000,C 90.000,E1 52.190} C_DIS
LIN {X 0.107,Y -533.299,Z 751.087,A 0.000,B 0.000,C 90.000,E1 51.618} C_DIS
LIN {X 0.092,Y -529.338,Z 751.084,A 0.000,B 0.000,C 90.000,E1 51.045} C_DIS
LIN {X -0.026,Y -524.903,Z 751.081,A 0.000,B 0.000,C 90.000,E1 50.481} C_DIS
LIN {X 0.244,Y -520.323,Z 751.077,A 0.000,B 0.000,C 90.000,E1 49.908} C_DIS
LIN {X 0.249,Y -515.270,Z 751.075,A 0.000,B 0.000,C 90.000,E1 49.380} C_DIS
LIN {X 0.152,Y -511.488,Z 751.072,A 0.000,B 0.000,C 90.000,E1 49.013} C_DIS
LIN {X -0.083,Y -505.686,Z 751.070,A 0.000,B 0.000,C 90.000,E1 48.528} C_DIS
LIN {X -0.173,Y -497.961,Z 751.066,A 0.000,B 0.000,C 90.000,E1 47.919} C_DIS
LIN {X -0.114,Y -493.136,Z 751.064,A 0.000,B 0.000,C 90.000,E1 47.553} C_DIS
LIN {X 0.099,Y -483.632,Z 751.060,A 0.000,B 0.000,C 90.000,E1 46.863} C_DIS
LIN {X 0.136,Y -467.281,Z 751.055,A 0.000,B 0.000,C 90.000,E1 45.810} C_DIS
LIN {X -0.079,Y -449.390,Z 751.048,A 0.000,B 0.000,C 90.000,E1 44.676} C_DIS
LIN {X -0.090,Y -425.271,Z 751.039,A 0.000,B 0.000,C 90.000,E1 43.014} C_DIS
LIN {X -0.091,Y -415.906,Z 751.035,A 0.000,B 0.000,C 90.000,E1 42.285} C_DIS
LIN {X 0.175,Y -412.128,Z 751.033,A 0.000,B 0.000,C 90.000,E1 41.919} C_DIS
LIN {X 0.146,Y -412.104,Z 751.033,A 0.000,B 0.000,C 90.000,E1 41.919} C_DIS
LIN {X 0.073,Y -406.176,Z 751.015,A 0.000,B 0.000,C 90.000,E1 38.669} C_DIS
LIN {X 0.107,Y -404.745,Z 751.011,A 0.000,B 0.000,C 90.000,E1 37.971} C_DIS
LIN {X -0.025,Y -401.450,Z 751.002,A 0.000,B 0.000,C 90.000,E1 36.423} C_DIS
LIN {X -0.106,Y -401.337,Z 751.000,A 0.000,B 0.000,C 90.000,E1 36.091} C_DIS
LIN {X -0.098,Y -401.801,Z 750.985,A 0.000,B 0.000,C 90.000,E1 33.293} C_DIS
LIN {X -0.083,Y -402.656,Z 750.971,A 0.000,B 0.000,C 90.000,E1 30.846} C_DIS
LIN {X -0.113,Y -403.911,Z 750.958,A 0.000,B 0.000,C 90.000,E1 28.409} C_DIS
LIN {X 0.131,Y -405.459,Z 750.942,A 0.000,B 0.000,C 90.000,E1 25.591} C_DIS
LIN {X -0.179,Y -407.233,Z 750.929,A 0.000,B 0.000,C 90.000,E1 23.206} C_DIS
LIN {X -0.115,Y -410.839,Z 750.908,A 0.000,B 0.000,C 90.000,E1 19.396} C_DIS
LIN {X 0.056,Y -414.206,Z 750.892,A 0.000,B 0.000,C 90.000,E1 16.622} C_DIS
LIN {X -0.100,Y -417.088,Z 750.881,A 0.000,B 0.000,C 90.000,E1 14.592} C_DIS
LIN {X 0.073,Y -420.727,Z 750.868,A 0.000,B 0.000,C 90.000,E1 12.187} C_DIS
LIN {X 0.111,Y -423.469,Z 750.858,A 0.000,B 0.000,C 90.000,E1 10.489} C_DIS
LIN {X -0.207,Y -426.681,Z 750.847,A 0.000,B 0.000,C 90.000,E1 8.511} C_DIS
LIN {X -0.101,Y -429.895,Z 750.836,A 0.000,B 0.000,C 90.000,E1 6.486} C_DIS
LIN {X 0.177,Y -434.446,Z 750.821,A 0.000,B 0.000,C 90.000,E1 3.784} C_DIS
LIN {X -0.105,Y -438.073,Z 750.810,A 0.000,B 0.000,C 90.000,E1 1.835} C_DIS
LIN {X 0.000,Y -441.537,Z 750.800,A 0.000,B 0.000,C 90.000,E1 360.000} C_DIS
LIN {X -0.217,Y -444.511,Z 750.792,A 0.000,B 0.000,C 90.000,E1 358.511} C_DIS
LIN {X 0.200,Y -448.673,Z 750.781,A 0.000,B 0.000,C 90.000,E1 356.502} C_DIS
LIN {X -0.073,Y -455.183,Z 750.765,A 0.000,B 0.000,C 90.000,E1 353.628} C_DIS
LIN {X 0.062,Y -458.813,Z 750.756,A 0.000,B 0.000,C 90.000,E1 352.008} C_DIS
LIN {X -0.185,Y -462.250,Z 750.747,A 0.000,B 0.000,C 90.000,E1 350.443} C_DIS
LIN {X 0.109,Y -464.212,Z 750.742,A 0.000,B 0.000,C 90.000,E1 349.454} C_DIS
LIN {X 0.036,Y -467.265,Z 750.733,A 0.000,B 0.000,C 90.000,E1 347.881} C_DIS
LIN {X 0.135,Y -471.973,Z 750.719,A 0.000,B 0.000,C 90.000,E1 345.353} C_DIS
LIN {X -0.102,Y -473.202,Z 750.715,A 0.000,B 0.000,C 90.000,E1 344.755} C_DIS
LIN {X 0.085,Y -475.681,Z 750.710,A 0.000,B 0.000,C 90.000,E1 343.795} C_DIS
LIN {X -0.121,Y -477.827,Z 750.707,A 0.000,B 0.000,C 90.000,E1 343.196} C_DIS
LIN {X -0.072,Y -480.042,Z 750.704,A 0.000,B 0.000,C 90.000,E1 342.725} C_DIS
LIN {X 0.154,Y -483.298,Z 750.701,A 0.000,B 0.000,C 90.000,E1 342.181} C_DIS
LIN {X -0.231,Y -487.096,Z 750.699,A 0.000,B 0.000,C 90.000,E1 341.764} C_DIS
LIN {X -0.230,Y -492.173,Z 750.696,A 0.000,B 0.000,C 90.000,E1 341.275} C_DIS
LIN {X -0.236,Y -499.933,Z 750.693,A 0.000,B 0.000,C 90.000,E1 340.678} C_DIS
LIN {X -0.007,Y -511.011,Z 750.688,A 0.000,B 0.000,C 90.000,E1 339.880} C_DIS
LIN {X -0.183,Y -526.958,Z 750.683,A 0.000,B 0.000,C 90.000,E1 338.901} C_DIS
LIN {X -0.096,Y -536.443,Z 750.680,A 0.000,B 0.000,C 90.000,E1 338.337} C_DIS
LIN {X -0.229,Y -544.042,Z 750.677,A 0.000,B 0.000,C 90.000,E1 337.847} C_DIS
LIN {X -0.113,Y -550.001,Z 750.674,A 0.000,B 0.000,C 90.000,E1 337.411} C_DIS
LIN {X 0.114,Y -555.580,Z 750.672,A 0.000,B 0.000,C 90.000,E1 336.922} C_DIS
LIN {X 0.022,Y -560.949,Z 750.669,A 0.000,B 0.000,C 90.000,E1 336.433} C_DIS
LIN {X -0.159,Y -567.240,Z 750.665,A 0.000,B 0.000,C 90.000,E1 335.793} C_DIS
LIN {X 0.091,Y -572.140,Z 750.662,A 0.000,B 0.000,C 90.000,E1 335.229} C_DIS
LIN {X 0.130,Y -579.181,Z 750.658,A 0.000,B 0.000,C 90.000,E1 334.409} C_DIS
LIN {X 0.177,Y -586.818,Z 750.653,A 0.000,B 0.000,C 90.000,E1 333.461} C_DIS
LIN {X 0.007,Y -594.991,Z 750.647,A 0.000,B 0.000,C 90.000,E1 332.410} C_DIS
LIN {X -0.330,Y -602.690,Z 750.641,A 0.000,B 0.000,C 90.000,E1 331.385} C_DIS
LIN {X -0.256,Y -609.141,Z 750.636,A 0.000,B 0.000,C 90.000,E1 330.461} C_DIS
LIN {X -0.084,Y -614.390,Z 750.631,A 0.000,B 0.000,C 90.000,E1 329.665} C_DIS
LIN {X 0.145,Y -619.413,Z 750.627,A 0.000,B 0.000,C 90.000,E1 328.869} C_DIS
LIN {X -0.109,Y -624.948,Z 750.622,A 0.000,B 0.000,C 90.000,E1 327.995} C_DIS
LIN {X 0.220,Y -628.752,Z 750.619,A 0.000,B 0.000,C 90.000,E1 327.327} C_DIS
LIN {X 0.416,Y -633.722,Z 750.614,A 0.000,B 0.000,C 90.000,E1 326.421} C_DIS
LIN {X -0.198,Y -639.026,Z 750.608,A 0.000,B 0.000,C 90.000,E1 325.468} C_DIS
LIN {X 0.117,Y -643.444,Z 750.603,A 0.000,B 0.000,C 90.000,E1 324.562} C_DIS
LIN {X -0.020,Y -648.206,Z 750.598,A 0.000,B 0.000,C 90.000,E1 323.577} C_DIS
LIN {X 0.291,Y -652.585,Z 750.592,A 0.000,B 0.000,C 90.000,E1 322.557} C_DIS
LIN {X 0.208,Y -655.796,Z 750.588,A 0.000,B 0.000,C 90.000,E1 321.823} C_DIS
LIN {X -0.299,Y -659.655,Z 750.583,A 0.000,B 0.000,C 90.000,E1 320.884} C_DIS
LIN {X 0.107,Y -662.438,Z 750.578,A 0.000,B 0.000,C 90.000,E1 320.114} C_DIS
LIN {X 0.107,Y -665.934,Z 750.573,A 0.000,B 0.000,C 90.000,E1 319.138} C_DIS
LIN {X 0.148,Y -668.426,Z 750.569,A 0.000,B 0.000,C 90.000,E1 318.405} C_DIS
LIN {X -0.274,Y -672.242,Z 750.562,A 0.000,B 0.000,C 90.000,E1 317.229} C_DIS
LIN {X 0.319,Y -675.810,Z 750.556,A 0.000,B 0.000,C 90.000,E1 315.972} C_DIS
LIN {X -0.030,Y -678.428,Z 750.550,A 0.000,B 0.000,C 90.000,E1 315.040} C_DIS
LIN {X -0.349,Y -680.769,Z 750.545,A 0.000,B 0.000,C 90.000,E1 314.109} C_DIS
LIN {X -0.112,Y -683.554,Z 750.538,A 0.000,B 0.000,C 90.000,E1 312.894} C_DIS
LIN {X 0.146,Y -685.590,Z 750.533,A 0.000,B 0.000,C 90.000,E1 311.919} C_DIS
LIN {X -0.405,Y -688.297,Z 750.525,A 0.000,B 0.000,C 90.000,E1 310.539} C_DIS
LIN {X -0.076,Y -689.789,Z 750.520,A 0.000,B 0.000,C 90.000,E1 309.564} C_DIS
LIN {X 0.208,Y -690.786,Z 750.516,A 0.000,B 0.000,C 90.000,E1 308.830} C_DIS
LIN {X 0.198,Y -692.277,Z 750.509,A 0.000,B 0.000,C 90.000,E1 307.649} C_DIS
LIN {X 0.142,Y -693.386,Z 750.504,A 0.000,B 0.000,C 90.000,E1 306.710} C_DIS
LIN {X -0.048,Y -694.671,Z 750.496,A 0.000,B 0.000,C 90.000,E1 305.311} C_DIS
LIN {X -0.210,Y -695.846,Z 750.488,A 0.000,B 0.000,C 90.000,E1 303.913} C_DIS
LIN {X 0.222,Y -696.951,Z 750.481,A 0.000,B 0.000,C 90.000,E1 302.467} C_DIS
LIN {X -0.049,Y -698.169,Z 750.471,A 0.000,B 0.000,C 90.000,E1 300.846} C_DIS
LIN {X 0.119,Y -698.554,Z 750.467,A 0.000,B 0.000,C 90.000,E1 300.129} C_DIS
LIN {X 0.216,Y -698.953,Z 750.461,A 0.000,B 0.000,C 90.000,E1 298.949} C_DIS
LIN {X -0.036,Y -699.410,Z 750.453,A 0.000,B 0.000,C 90.000,E1 297.564} C_DIS
LIN {X 0.155,Y -700.445,Z 750.440,A 0.000,B 0.000,C 90.000,E1 295.207} C_DIS
LIN {X -0.233,Y -700.531,Z 750.438,A 0.000,B 0.000,C 90.000,E1 294.771} C_DIS
LIN {X 0.037,Y -700.347,Z 750.436,A 0.000,B 0.000,C 90.000,E1 294.515} C_DIS
LIN {X -0.349,Y -699.622,Z 750.434,A 0.000,B 0.000,C 90.000,E1 294.079} C_DIS
LIN {X -0.080,Y -698.700,Z 750.432,A 0.000,B 0.000,C 90.000,E1 293.823} C_DIS
LIN {X 0.165,Y -696.040,Z 750.430,A 0.000,B 0.000,C 90.000,E1 293.334} C_DIS
LIN {X 0.292,Y -695.098,Z 750.429,A 0.000,B 0.000,C 90.000,E1 293.206} C_DIS
LIN {X -0.220,Y -693.695,Z 750.428,A 0.000,B 0.000,C 90.000,E1 293.131} C_DIS
LIN {X -0.020,Y -689.759,Z 750.427,A 0.000,B 0.000,C 90.000,E1 292.898} C_DIS
LIN {X 0.201,Y -686.677,Z 750.426,A 0.000,B 0.000,C 90.000,E1 292.717} C_DIS
LIN {X 0.117,Y -684.752,Z 750.426,A 0.000,B 0.000,C 90.000,E1 292.642} C_DIS
LIN {X -0.338,Y -676.168,Z 750.425,A 0.000,B 0.000,C 90.000,E1 292.461} C_DIS
LIN {X 0.233,Y -667.404,Z 750.424,A 0.000,B 0.000,C 90.000,E1 292.280} C_DIS
LIN {X -0.217,Y -657.928,Z 750.423,A 0.000,B 0.000,C 90.000,E1 292.206} C_DIS
LIN {X 0.149,Y -647.790,Z 750.422,A 0.000,B 0.000,C 90.000,E1 292.025} C_DIS
LIN {X 0.152,Y -638.150,Z 750.422,A 0.000,B 0.000,C 90.000,E1 291.844} C_DIS
LIN {X 0.229,Y -624.749,Z 750.420,A 0.000,B 0.000,C 90.000,E1 291.535} C_DIS
LIN {X 0.250,Y -607.585,Z 750.417,A 0.000,B 0.000,C 90.000,E1 291.099} C_DIS
LIN {X 0.004,Y -574.328,Z 750.412,A 0.000,B 0.000,C 90.000,E1 290.174} C_DIS
LIN {X -0.081,Y -566.962,Z 750.411,A 0.000,B 0.000,C 90.000,E1 289.993} C_DIS
LIN {X -0.047,Y -560.732,Z 750.410,A 0.000,B 0.000,C 90.000,E1 289.758} C_DIS
LIN {X -0.221,Y -557.132,Z 750.409,A 0.000,B 0.000,C 90.000,E1 289.577} C_DIS
LIN {X -0.100,Y -555.770,Z 750.408,A 0.000,B 0.000,C 90.000,E1 289.396} C_DIS
LIN {X -0.142,Y -555.757,Z 750.408,A 0.000,B 0.000,C 90.000,E1 289.396} C_DIS
LIN {X 0.325,Y -555.029,Z 750.406,A 0.000,B 0.000,C 90.000,E1 288.960} C_DIS
LIN {X -0.107,Y -554.669,Z 750.402,A 0.000,B 0.000,C 90.000,E1 288.308} C_DIS
LIN {X 0.036,Y -554.422,Z 750.397,A 0.000,B 0.000,C 90.000,E1 287.457} C_DIS
LIN {X -0.020,Y -553.793,Z 750.388,A 0.000,B 0.000,C 90.000,E1 285.788} C_DIS
LIN {X -0.090,Y -553.216,Z 750.378,A 0.000,B 0.000,C 90.000,E1 284.120} C_DIS
LIN {X -0.024,Y -552.693,Z 750.371,A 0.000,B 0.000,C 90.000,E1 282.715} C_DIS
LIN {X -0.257,Y -552.129,Z 750.360,A 0.000,B 0.000,C 90.000,E1 280.782} C_DIS
LIN {X -0.071,Y -551.346,Z 750.349,A 0.000,B 0.000,C 90.000,E1 278.803} C_DIS
LIN {X 0.001,Y -550.416,Z 750.338,A 0.000,B 0.000,C 90.000,E1 276.834} C_DIS
LIN {X 0.243,Y -550.058,Z 750.333,A 0.000,B 0.000,C 90.000,E1 275.967} C_DIS
LIN {X 0.013,Y -549.227,Z 750.326,A 0.000,B 0.000,C 90.000,E1 274.588} C_DIS
LIN {X -0.140,Y -548.162,Z 750.315,A 0.000,B 0.000,C 90.000,E1 272.636} C_DIS
LIN {X 0.113,Y -547.412,Z 750.307,A 0.000,B 0.000,C 90.000,E1 271.203} C_DIS
LIN {X -0.205,Y -546.633,Z 750.299,A 0.000,B 0.000,C 90.000,E1 269.828} C_DIS
LIN {X 0.006,Y -545.667,Z 750.291,A 0.000,B 0.000,C 90.000,E1 268.396} C_DIS
LIN {X -0.239,Y -544.405,Z 750.280,A 0.000,B 0.000,C 90.000,E1 266.445} C_DIS
LIN {X -0.018,Y -543.503,Z 750.272,A 0.000,B 0.000,C 90.000,E1 265.008} C_DIS
LIN {X 0.254,Y -542.322,Z 750.263,A 0.000,B 0.000,C 90.000,E1 263.280} C_DIS
LIN {X -0.127,Y -541.661,Z 750.258,A 0.000,B 0.000,C 90.000,E1 262.470} C_DIS
LIN {X 0.164,Y -540.227,Z 750.249,A 0.000,B 0.000,C 90.000,E1 260.735} C_DIS
LIN {X -0.172,Y -539.281,Z 750.242,A 0.000,B 0.000,C 90.000,E1 259.634} C_DIS
LIN {X 0.238,Y -537.920,Z 750.233,A 0.000,B 0.000,C 90.000,E1 257.881} C_DIS
LIN {X -0.096,Y -537.162,Z 750.228,A 0.000,B 0.000,C 90.000,E1 257.061} C_DIS
LIN {X -0.199,Y -535.860,Z 750.220,A 0.000,B 0.000,C 90.000,E1 255.644} C_DIS
LIN {X -0.140,Y -534.004,Z 750.211,A 0.000,B 0.000,C 90.000,E1 253.921} C_DIS
LIN {X 0.030,Y -532.042,Z 750.201,A 0.000,B 0.000,C 90.000,E1 252.181} C_DIS
LIN {X -0.052,Y -530.819,Z 750.195,A 0.000,B 0.000,C 90.000,E1 251.040} C_DIS
LIN {X -0.106,Y -528.480,Z 750.185,A 0.000,B 0.000,C 90.000,E1 249.316} C_DIS
LIN {X 0.113,Y -526.438,Z 750.177,A 0.000,B 0.000,C 90.000,E1 247.847} C_DIS
LIN {X 0.168,Y -523.832,Z 750.167,A 0.000,B 0.000,C 90.000,E1 246.102} C_DIS
LIN {X -0.147,Y -521.974,Z 750.161,A 0.000,B 0.000,C 90.000,E1 244.973} C_DIS
LIN {X 0.202,Y -520.072,Z 750.154,A 0.000,B 0.000,C 90.000,E1 243.768} C_DIS
LIN {X -0.078,Y -518.562,Z 750.150,A 0.000,B 0.000,C 90.000,E1 242.922} C_DIS
LIN {X 0.116,Y -515.851,Z 750.141,A 0.000,B 0.000,C 90.000,E1 241.435} C_DIS
LIN {X 0.153,Y -512.421,Z 750.132,A 0.000,B 0.000,C 90.000,E1 239.665} C_DIS
LIN {X -0.309,Y -510.099,Z 750.125,A 0.000,B 0.000,C 90.000,E1 238.535} C_DIS
LIN {X 0.264,Y -508.323,Z 750.120,A 0.000,B 0.000,C 90.000,E1 237.582} C_DIS
LIN {X 0.115,Y -506.485,Z 750.115,A 0.000,B 0.000,C 90.000,E1 236.707} C_DIS
LIN {X 0.116,Y -503.811,Z 750.109,A 0.000,B 0.000,C 90.000,E1 235.515} C_DIS
LIN {X -0.033,Y -500.311,Z 750.100,A 0.000,B 0.000,C 90.000,E1 234.036} C_DIS
LIN {X -0.123,Y -497.358,Z 750.094,A 0.000,B 0.000,C 90.000,E1 232.844} C_DIS
LIN {X -0.085,Y -492.047,Z 750.082,A 0.000,B 0.000,C 90.000,E1 230.723} C_DIS
LIN {X 0.087,Y -485.636,Z 750.067,A 0.000,B 0.000,C 90.000,E1 227.957} C_DIS
LIN {X -0.087,Y -481.668,Z 750.056,A 0.000,B 0.000,C 90.000,E1 226.134} C_DIS
LIN {X 0.107,Y -477.084,Z 750.044,A 0.000,B 0.000,C 90.000,E1 223.947} C_DIS
LIN {X 0.094,Y -473.081,Z 750.034,A 0.000,B 0.000,C 90.000,E1 222.081} C_DIS
LIN {X 0.053,Y -471.030,Z 750.029,A 0.000,B 0.000,C 90.000,E1 221.148} C_DIS
LIN {X 0.180,Y -467.545,Z 750.020,A 0.000,B 0.000,C 90.000,E1 219.564} C_DIS
LIN {X 0.102,Y -462.799,Z 750.008,A 0.000,B 0.000,C 90.000,E1 217.363} C_DIS
LIN {X 0.090,Y -457.530,Z 749.994,A 0.000,B 0.000,C 90.000,E1 214.818} C_DIS
LIN {X 0.030,Y -452.474,Z 749.979,A 0.000,B 0.000,C 90.000,E1 212.260} C_DIS
LIN {X 0.020,Y -448.234,Z 749.967,A 0.000,B 0.000,C 90.000,E1 210.001} C_DIS
LIN {X 0.093,Y -445.796,Z 749.960,A 0.000,B 0.000,C 90.000,E1 208.693} C_DIS
LIN {X 0.127,Y -443.468,Z 749.952,A 0.000,B 0.000,C 90.000,E1 207.385} C_DIS
LIN {X -0.201,Y -439.727,Z 749.941,A 0.000,B 0.000,C 90.000,E1 205.463} C_DIS
LIN {X 0.163,Y -436.647,Z 749.932,A 0.000,B 0.000,C 90.000,E1 203.770} C_DIS
LIN {X -0.107,Y -433.560,Z 749.923,A 0.000,B 0.000,C 90.000,E1 202.153} C_DIS
LIN {X 0.146,Y -431.061,Z 749.916,A 0.000,B 0.000,C 90.000,E1 200.791} C_DIS
LIN {X 0.211,Y -427.294,Z 749.905,A 0.000,B 0.000,C 90.000,E1 198.779} C_DIS
LIN {X -0.145,Y -424.099,Z 749.895,A 0.000,B 0.000,C 90.000,E1 197.149} C_DIS
LIN {X -0.220,Y -420.125,Z 749.884,A 0.000,B 0.000,C 90.000,E1 195.134} C_DIS
LIN {X 0.076,Y -415.745,Z 749.871,A 0.000,B 0.000,C 90.000,E1 192.715} C_DIS
LIN {X 0.073,Y -412.750,Z 749.861,A 0.000,B 0.000,C 90.000,E1 191.007} C_DIS
LIN {X -0.156,Y -409.855,Z 749.852,A 0.000,B 0.000,C 90.000,E1 189.321} C_DIS
LIN {X -0.067,Y -405.808,Z 749.838,A 0.000,B 0.000,C 90.000,E1 186.891} C_DIS
LIN {X -0.175,Y -402.523,Z 749.827,A 0.000,B 0.000,C 90.000,E1 184.821} C_DIS
LIN {X 0.113,Y -400.511,Z 749.819,A 0.000,B 0.000,C 90.000,E1 183.383} C_DIS
LIN {X 0.080,Y -396.331,Z 749.801,A 0.000,B 0.000,C 90.000,E1 180.229} C_DIS
LIN {X -0.038,Y -393.209,Z 749.786,A 0.000,B 0.000,C 90.000,E1 177.421} C_DIS
LIN {X 0.053,Y -389.832,Z 749.766,A 0.000,B 0.000,C 90.000,E1 173.856} C_DIS
LIN {X 0.012,Y -387.428,Z 749.742,A 0.000,B 0.000,C 90.000,E1 169.577} C_DIS
LIN {X 0.075,Y -386.241,Z 749.728,A 0.000,B 0.000,C 90.000,E1 167.061} C_DIS
LIN {X -0.025,Y -385.479,Z 749.718,A 0.000,B 0.000,C 90.000,E1 165.283} C_DIS
LIN {X -0.099,Y -384.736,Z 749.704,A 0.000,B 0.000,C 90.000,E1 162.779} C_DIS
LIN {X 0.064,Y -384.003,Z 749.686,A 0.000,B 0.000,C 90.000,E1 159.518} C_DIS
LIN {X 0.066,Y -383.637,Z 749.672,A 0.000,B 0.000,C 90.000,E1 156.997} C_DIS
LIN {X 0.168,Y -383.537,Z 749.658,A 0.000,B 0.000,C 90.000,E1 154.460} C_DIS
LIN {X -0.067,Y -386.630,Z 749.620,A 0.000,B 0.000,C 90.000,E1 147.661} C_DIS
LIN {X 0.069,Y -388.989,Z 749.606,A 0.000,B 0.000,C 90.000,E1 145.135} C_DIS
LIN {X 0.087,Y -392.494,Z 749.593,A 0.000,B 0.000,C 90.000,E1 142.637} C_DIS
LIN {X -0.130,Y -395.380,Z 749.585,A 0.000,B 0.000,C 90.000,E1 141.251} C_DIS
LIN {X 0.055,Y -397.317,Z 749.581,A 0.000,B 0.000,C 90.000,E1 140.517} C_DIS
LIN {X -0.153,Y -398.522,Z 749.579,A 0.000,B 0.000,C 90.000,E1 140.194} C_DIS
LIN {X -0.102,Y -400.274,Z 749.576,A 0.000,B 0.000,C 90.000,E1 139.747} C_DIS
LIN {X 0.101,Y -403.134,Z 749.573,A 0.000,B 0.000,C 90.000,E1 139.138} C_DIS
LIN {X 0.008,Y -404.139,Z 749.572,A 0.000,B 0.000,C 90.000,E1 138.976} C_DIS
LIN {X 0.143,Y -407.961,Z 749.569,A 0.000,B 0.000,C 90.000,E1 138.405} C_DIS
LIN {X 0.071,Y -412.660,Z 749.566,A 0.000,B 0.000,C 90.000,E1 137.838} C_DIS
LIN {X 0.043,Y -425.084,Z 749.559,A 0.000,B 0.000,C 90.000,E1 136.539} C_DIS
LIN {X 0.104,Y -432.389,Z 749.555,A 0.000,B 0.000,C 90.000,E1 135.810} C_DIS
LIN {X 0.195,Y -445.265,Z 749.547,A 0.000,B 0.000,C 90.000,E1 134.514} C_DIS
LIN {X -0.081,Y -455.166,Z 749.542,A 0.000,B 0.000,C 90.000,E1 133.542} C_DIS
LIN {X -0.142,Y -461.849,Z 749.538,A 0.000,B 0.000,C 90.000,E1 132.852} C_DIS
LIN {X 0.035,Y -469.992,Z 749.533,A 0.000,B 0.000,C 90.000,E1 131.962} C_DIS
LIN {X 0.192,Y -479.399,Z 749.527,A 0.000,B 0.000,C 90.000,E1 130.906} C_DIS
LIN {X 0.011,Y -485.870,Z 749.523,A 0.000,B 0.000,C 90.000,E1 130.172} C_DIS
LIN {X 0.022,Y -491.970,Z 749.519,A 0.000,B 0.000,C 90.000,E1 129.439} C_DIS
LIN {X 0.283,Y -496.567,Z 749.516,A 0.000,B 0.000,C 90.000,E1 128.830} C_DIS
LIN {X 0.131,Y -501.994,Z 749.512,A 0.000,B 0.000,C 90.000,E1 128.096} C_DIS
LIN {X 0.106,Y -505.226,Z 749.509,A 0.000,B 0.000,C 90.000,E1 127.649} C_DIS
LIN {X 0.000,Y -510.122,Z 749.505,A 0.000,B 0.000,C 90.000,E1 126.916} C_DIS
LIN {X 0.041,Y -514.637,Z 749.501,A 0.000,B 0.000,C 90.000,E1 126.171} C_DIS
LIN {X 0.016,Y -519.008,Z 749.497,A 0.000,B 0.000,C 90.000,E1 125.438} C_DIS
LIN {X -0.045,Y -520.709,Z 749.495,A 0.000,B 0.000,C 90.000,E1 125.152} C_DIS
LIN {X -0.102,Y -526.499,Z 749.489,A 0.000,B 0.000,C 90.000,E1 123.992} C_DIS
LIN {X -0.301,Y -528.534,Z 749.486,A 0.000,B 0.000,C 90.000,E1 123.579} C_DIS
LIN {X -0.104,Y -534.338,Z 749.479,A 0.000,B 0.000,C 90.000,E1 122.260} C_DIS
LIN {X -0.105,Y -538.535,Z 749.474,A 0.000,B 0.000,C 90.000,E1 121.258} C_DIS
LIN {X 0.077,Y -541.896,Z 749.469,A 0.000,B 0.000,C 90.000,E1 120.384} C_DIS
LIN {X 0.285,Y -544.009,Z 749.466,A 0.000,B 0.000,C 90.000,E1 119.795} C_DIS
LIN {X 0.258,Y -547.026,Z 749.461,A 0.000,B 0.000,C 90.000,E1 118.949} C_DIS
LIN {X 0.268,Y -549.884,Z 749.456,A 0.000,B 0.000,C 90.000,E1 118.103} C_DIS
LIN {X 0.306,Y -552.612,Z 749.452,A 0.000,B 0.000,C 90.000,E1 117.257} C_DIS
LIN {X 0.124,Y -555.143,Z 749.447,A 0.000,B 0.000,C 90.000,E1 116.437} C_DIS
LIN {X 0.214,Y -557.231,Z 749.442,A 0.000,B 0.000,C 90.000,E1 115.591} C_DIS
LIN {X 0.082,Y -559.027,Z 749.438,A 0.000,B 0.000,C 90.000,E1 114.771} C_DIS
LIN {X 0.274,Y -560.957,Z 749.432,A 0.000,B 0.000,C 90.000,E1 113.643} C_DIS
LIN {X -0.241,Y -562.651,Z 749.425,A 0.000,B 0.000,C 90.000,E1 112.589} C_DIS
LIN {X -0.084,Y -564.926,Z 749.416,A 0.000,B 0.000,C 90.000,E1 110.918} C_DIS
LIN {X -0.025,Y -566.405,Z 749.410,A 0.000,B 0.000,C 90.000,E1 109.812} C_DIS
LIN {X -0.188,Y -568.406,Z 749.401,A 0.000,B 0.000,C 90.000,E1 108.181} C_DIS
LIN {X 0.233,Y -570.216,Z 749.392,A 0.000,B 0.000,C 90.000,E1 106.496} C_DIS
LIN {X 0.161,Y -572.260,Z 749.381,A 0.000,B 0.000,C 90.000,E1 104.592} C_DIS
LIN {X -0.013,Y -574.279,Z 749.371,A 0.000,B 0.000,C 90.000,E1 102.703} C_DIS
LIN {X -0.027,Y -576.056,Z 749.362,A 0.000,B 0.000,C 90.000,E1 101.074} C_DIS
LIN {X 0.011,Y -577.729,Z 749.353,A 0.000,B 0.000,C 90.000,E1 99.443} C_DIS
LIN {X 0.213,Y -578.787,Z 749.346,A 0.000,B 0.000,C 90.000,E1 98.341} C_DIS
LIN {X -0.148,Y -580.508,Z 749.336,A 0.000,B 0.000,C 90.000,E1 96.486} C_DIS
LIN {X 0.168,Y -581.605,Z 749.328,A 0.000,B 0.000,C 90.000,E1 95.106} C_DIS
LIN {X -0.072,Y -582.614,Z 749.321,A 0.000,B 0.000,C 90.000,E1 93.784} C_DIS
LIN {X -0.154,Y -583.739,Z 749.312,A 0.000,B 0.000,C 90.000,E1 92.178} C_DIS
LIN {X 0.004,Y -584.451,Z 749.306,A 0.000,B 0.000,C 90.000,E1 91.088} C_DIS
LIN {X -0.053,Y -585.285,Z 749.297,A 0.000,B 0.000,C 90.000,E1 89.484} C_DIS
LIN {X -0.080,Y -585.888,Z 749.288,A 0.000,B 0.000,C 90.000,E1 87.879} C_DIS
LIN {X -0.097,Y -586.400,Z 749.279,A 0.000,B 0.000,C 90.000,E1 86.274} C_DIS
LIN {X 0.145,Y -586.610,Z 749.273,A 0.000,B 0.000,C 90.000,E1 85.179} C_DIS
LIN {X -0.007,Y -586.819,Z 749.266,A 0.000,B 0.000,C 90.000,E1 83.856} C_DIS
LIN {X -0.092,Y -586.906,Z 749.258,A 0.000,B 0.000,C 90.000,E1 82.527} C_DIS
LIN {X 0.074,Y -586.865,Z 749.250,A 0.000,B 0.000,C 90.000,E1 80.905} C_DIS
LIN {X 0.078,Y -586.676,Z 749.242,A 0.000,B 0.000,C 90.000,E1 79.567} C_DIS
LIN {X -0.251,Y -586.238,Z 749.233,A 0.000,B 0.000,C 90.000,E1 77.993} C_DIS
LIN {X 0.172,Y -585.861,Z 749.227,A 0.000,B 0.000,C 90.000,E1 76.881} C_DIS
LIN {X -0.166,Y -585.260,Z 749.220,A 0.000,B 0.000,C 90.000,E1 75.574} C_DIS
LIN {X 0.056,Y -584.593,Z 749.212,A 0.000,B 0.000,C 90.000,E1 74.212} C_DIS
LIN {X -0.305,Y -583.824,Z 749.205,A 0.000,B 0.000,C 90.000,E1 72.906} C_DIS
LIN {X -0.178,Y -583.080,Z 749.199,A 0.000,B 0.000,C 90.000,E1 71.819} C_DIS
LIN {X 0.341,Y -582.096,Z 749.191,A 0.000,B 0.000,C 90.000,E1 70.423} C_DIS
LIN {X 0.292,Y -580.979,Z 749.184,A 0.000,B 0.000,C 90.000,E1 69.082} C_DIS
LIN {X -0.323,Y -579.670,Z 749.177,A 0.000,B 0.000,C 90.000,E1 67.794} C_DIS
LIN {X 0.165,Y -578.522,Z 749.171,A 0.000,B 0.000,C 90.000,E1 66.666} C_DIS
LIN {X -0.125,Y -577.211,Z 749.164,A 0.000,B 0.000,C 90.000,E1 65.613} C_DIS
LIN {X -0.200,Y -575.711,Z 749.158,A 0.000,B 0.000,C 90.000,E1 64.537} C_DIS
LIN {X -0.039,Y -574.102,Z 749.152,A 0.000,B 0.000,C 90.000,E1 63.435} C_DIS
LIN {X 0.003,Y -572.677,Z 749.148,A 0.000,B 0.000,C 90.000,E1 62.615} C_DIS
LIN {X 0.288,Y -571.135,Z 749.143,A 0.000,B 0.000,C 90.000,E1 61.769} C_DIS
LIN {X -0.115,Y -568.699,Z 749.137,A 0.000,B 0.000,C 90.000,E1 60.717} C_DIS
LIN {X 0.125,Y -566.699,Z 749.133,A 0.000,B 0.000,C 90.000,E1 59.871} C_DIS
LIN {X -0.050,Y -563.765,Z 749.127,A 0.000,B 0.000,C 90.000,E1 58.791} C_DIS
LIN {X 0.123,Y -561.314,Z 749.122,A 0.000,B 0.000,C 90.000,E1 57.946} C_DIS
LIN {X 0.087,Y -558.648,Z 749.117,A 0.000,B 0.000,C 90.000,E1 57.120} C_DIS
LIN {X 0.177,Y -553.595,Z 749.110,A 0.000,B 0.000,C 90.000,E1 55.722} C_DIS
LIN {X 0.065,Y -550.115,Z 749.105,A 0.000,B 0.000,C 90.000,E1 54.895} C_DIS
LIN {X 0.043,Y -546.927,Z 749.101,A 0.000,B 0.000,C 90.000,E1 54.196} C_DIS
LIN {X -0.010,Y -543.366,Z 749.097,A 0.000,B 0.000,C 90.000,E1 53.497} C_DIS
LIN {X 0.227,Y -539.509,Z 749.093,A 0.000,B 0.000,C 90.000,E1 52.763} C_DIS
LIN {X 0.092,Y -537.076,Z 749.091,A 0.000,B 0.000,C 90.000,E1 52.351} C_DIS
LIN {X -0.136,Y -532.528,Z 749.087,A 0.000,B 0.000,C 90.000,E1 51.662} C_DIS
LIN {X -0.139,Y -528.486,Z 749.084,A 0.000,B 0.000,C 90.000,E1 51.090} C_DIS
LIN {X -0.086,Y -524.015,Z 749.081,A 0.000,B 0.000,C 90.000,E1 50.517} C_DIS
LIN {X 0.141,Y -520.428,Z 749.078,A 0.000,B 0.000,C 90.000,E1 50.070} C_DIS
LIN {X -0.180,Y -514.998,Z 749.075,A 0.000,B 0.000,C 90.000,E1 49.542} C_DIS
LIN {X -0.069,Y -509.585,Z 749.072,A 0.000,B 0.000,C 90.000,E1 49.013} C_DIS
LIN {X 0.084,Y -505.123,Z 749.070,A 0.000,B 0.000,C 90.000,E1 48.609} C_DIS
LIN {X -0.148,Y -495.978,Z 749.066,A 0.000,B 0.000,C 90.000,E1 47.919} C_DIS
LIN {X -0.077,Y -486.365,Z 749.062,A 0.000,B 0.000,C 90.000,E1 47.229} C_DIS
LIN {X -0.113,Y -481.346,Z 749.061,A 0.000,B 0.000,C 90.000,E1 46.905} C_DIS
LIN {X -0.107,Y -466.787,Z 749.055,A 0.000,B 0.000,C 90.000,E1 45.972} C_DIS
LIN {X 0.028,Y -448.887,Z 749.049,A 0.000,B 0.000,C 90.000,E1 44.798} C_DIS
LIN {X 0.076,Y -424.915,Z 749.040,A 0.000,B 0.000,C 90.000,E1 43.137} C_DIS
LIN {X 0.118,Y -417.083,Z 749.036,A 0.000,B 0.000,C 90.000,E1 42.528} C_DIS
LIN {X -0.024,Y -412.594,Z 749.034,A 0.000,B 0.000,C 90.000,E1 42.162} C_DIS
LIN {X -0.053,Y -412.550,Z 749.034,A 0.000,B 0.000,C 90.000,E1 42.162} C_DIS
LIN {X -0.060,Y -406.076,Z 749.015,A 0.000,B 0.000,C 90.000,E1 38.624} C_DIS
LIN {X -0.069,Y -403.104,Z 749.007,A 0.000,B 0.000,C 90.000,E1 37.237} C_DIS
LIN {X 0.188,Y -401.670,Z 749.003,A 0.000,B 0.000,C 90.000,E1 36.503} C_DIS
LIN {X 0.095,Y -402.111,Z 748.986,A 0.000,B 0.000,C 90.000,E1 33.372} C_DIS
LIN {X -0.082,Y -403.321,Z 748.968,A 0.000,B 0.000,C 90.000,E1 30.256} C_DIS
LIN {X 0.009,Y -404.363,Z 748.956,A 0.000,B 0.000,C 90.000,E1 28.153} C_DIS
LIN {X 0.112,Y -405.555,Z 748.945,A 0.000,B 0.000,C 90.000,E1 26.052} C_DIS
LIN {X 0.083,Y -407.517,Z 748.929,A 0.000,B 0.000,C 90.000,E1 23.281} C_DIS
LIN {X -0.061,Y -410.000,Z 748.914,A 0.000,B 0.000,C 90.000,E1 20.536} C_DIS
LIN {X -0.068,Y -412.676,Z 748.901,A 0.000,B 0.000,C 90.000,E1 18.127} C_DIS
LIN {X -0.136,Y -415.345,Z 748.889,A 0.000,B 0.000,C 90.000,E1 16.079} C_DIS
LIN {X 0.029,Y -418.284,Z 748.878,A 0.000,B 0.000,C 90.000,E1 14.008} C_DIS
LIN {X -0.167,Y -421.968,Z 748.865,A 0.000,B 0.000,C 90.000,E1 11.658} C_DIS
LIN {X -0.194,Y -424.139,Z 748.857,A 0.000,B 0.000,C 90.000,E1 10.310} C_DIS
LIN {X -0.083,Y -427.348,Z 748.846,A 0.000,B 0.000,C 90.000,E1 8.276} C_DIS
LIN {X -0.120,Y -430.025,Z 748.837,A 0.000,B 0.000,C 90.000,E1 6.606} C_DIS
LIN {X 0.095,Y -433.942,Z 748.824,A 0.000,B 0.000,C 90.000,E1 4.245} C_DIS
LIN {X -0.177,Y -437.516,Z 748.813,A 0.000,B 0.000,C 90.000,E1 2.293} C_DIS
LIN {X 0.052,Y -441.250,Z 748.802,A 0.000,B 0.000,C 90.000,E1 0.286} C_DIS
LIN {X 0.207,Y -446.815,Z 748.786,A 0.000,B 0.000,C 90.000,E1 357.478} C_DIS
LIN {X -0.213,Y -450.996,Z 748.775,A 0.000,B 0.000,C 90.000,E1 355.584} C_DIS
LIN {X -0.055,Y -455.386,Z 748.765,A 0.000,B 0.000,C 90.000,E1 353.628} C_DIS
LIN {X 0.084,Y -459.012,Z 748.756,A 0.000,B 0.000,C 90.000,E1 352.008} C_DIS
LIN {X 0.053,Y -461.780,Z 748.749,A 0.000,B 0.000,C 90.000,E1 350.735} C_DIS
LIN {X 0.137,Y -464.385,Z 748.742,A 0.000,B 0.000,C 90.000,E1 349.454} C_DIS
LIN {X -0.196,Y -466.818,Z 748.734,A 0.000,B 0.000,C 90.000,E1 348.229} C_DIS
LIN {X 0.060,Y -469.146,Z 748.728,A 0.000,B 0.000,C 90.000,E1 346.937} C_DIS
LIN {X -0.115,Y -473.971,Z 748.714,A 0.000,B 0.000,C 90.000,E1 344.448} C_DIS
LIN {X -0.048,Y -476.478,Z 748.708,A 0.000,B 0.000,C 90.000,E1 343.504} C_DIS
LIN {X -0.250,Y -478.704,Z 748.705,A 0.000,B 0.000,C 90.000,E1 342.906} C_DIS
LIN {X 0.019,Y -480.990,Z 748.702,A 0.000,B 0.000,C 90.000,E1 342.417} C_DIS
LIN {X -0.143,Y -482.841,Z 748.701,A 0.000,B 0.000,C 90.000,E1 342.127} C_DIS
LIN {X -0.033,Y -485.461,Z 748.699,A 0.000,B 0.000,C 90.000,E1 341.764} C_DIS
LIN {X -0.031,Y -488.086,Z 748.697,A 0.000,B 0.000,C 90.000,E1 341.456} C_DIS
LIN {X -0.206,Y -494.245,Z 748.694,A 0.000,B 0.000,C 90.000,E1 340.913} C_DIS
LIN {X 0.167,Y -504.326,Z 748.690,A 0.000,B 0.000,C 90.000,E1 340.115} C_DIS
LIN {X -0.042,Y -515.559,Z 748.686,A 0.000,B 0.000,C 90.000,E1 339.390} C_DIS
LIN {X 0.171,Y -536.486,Z 748.679,A 0.000,B 0.000,C 90.000,E1 338.103} C_DIS
LIN {X 0.215,Y -545.722,Z 748.675,A 0.000,B 0.000,C 90.000,E1 337.486} C_DIS
LIN {X -0.076,Y -548.588,Z 748.674,A 0.000,B 0.000,C 90.000,E1 337.305} C_DIS
LIN {X -0.012,Y -553.981,Z 748.672,A 0.000,B 0.000,C 90.000,E1 336.869} C_DIS
LIN {X -0.169,Y -559.283,Z 748.669,A 0.000,B 0.000,C 90.000,E1 336.410} C_DIS
LIN {X 0.062,Y -564.442,Z 748.666,A 0.000,B 0.000,C 90.000,E1 335.869} C_DIS
LIN {X -0.293,Y -570.707,Z 748.662,A 0.000,B 0.000,C 90.000,E1 335.229} C_DIS
LIN {X -0.194,Y -577.774,Z 748.658,A 0.000,B 0.000,C 90.000,E1 334.409} C_DIS
LIN {X -0.037,Y -583.338,Z 748.654,A 0.000,B 0.000,C 90.000,E1 333.717} C_DIS
LIN {X -0.089,Y -588.672,Z 748.650,A 0.000,B 0.000,C 90.000,E1 333.050} C_DIS
LIN {X 0.068,Y -595.840,Z 748.645,A 0.000,B 0.000,C 90.000,E1 332.103} C_DIS
LIN {X 0.027,Y -603.564,Z 748.639,A 0.000,B 0.000,C 90.000,E1 331.051} C_DIS
LIN {X 0.094,Y -610.903,Z 748.633,A 0.000,B 0.000,C 90.000,E1 329.999} C_DIS
LIN {X -0.272,Y -617.771,Z 748.628,A 0.000,B 0.000,C 90.000,E1 328.997} C_DIS
LIN {X -0.023,Y -624.199,Z 748.622,A 0.000,B 0.000,C 90.000,E1 327.946} C_DIS
LIN {X 0.110,Y -629.496,Z 748.617,A 0.000,B 0.000,C 90.000,E1 327.041} C_DIS
LIN {X -0.043,Y -633.737,Z 748.613,A 0.000,B 0.000,C 90.000,E1 326.294} C_DIS
LIN {X 0.212,Y -638.460,Z 748.608,A 0.000,B 0.000,C 90.000,E1 325.388} C_DIS
LIN {X 0.139,Y -642.328,Z 748.604,A 0.000,B 0.000,C 90.000,E1 324.642} C_DIS
LIN {X -0.108,Y -648.342,Z 748.597,A 0.000,B 0.000,C 90.000,E1 323.417} C_DIS
LIN {X 0.283,Y -651.696,Z 748.593,A 0.000,B 0.000,C 90.000,E1 322.637} C_DIS
LIN {X 0.191,Y -654.949,Z 748.589,A 0.000,B 0.000,C 90.000,E1 321.904} C_DIS
LIN {X 0.086,Y -658.895,Z 748.583,A 0.000,B 0.000,C 90.000,E1 320.928} C_DIS
LIN {X 0.069,Y -661.740,Z 748.579,A 0.000,B 0.000,C 90.000,E1 320.194} C_DIS
LIN {X 0.044,Y -666.133,Z 748.572,A 0.000,B 0.000,C 90.000,E1 318.976} C_DIS
LIN {X 0.090,Y -667.859,Z 748.569,A 0.000,B 0.000,C 90.000,E1 318.485} C_DIS
LIN {X -0.342,Y -671.735,Z 748.563,A 0.000,B 0.000,C 90.000,E1 317.310} C_DIS
LIN {X 0.242,Y -675.353,Z 748.556,A 0.000,B 0.000,C 90.000,E1 316.053} C_DIS
LIN {X 0.366,Y -678.032,Z 748.551,A 0.000,B 0.000,C 90.000,E1 315.081} C_DIS
LIN {X -0.003,Y -679.912,Z 748.547,A 0.000,B 0.000,C 90.000,E1 314.393} C_DIS
LIN {X 0.294,Y -683.281,Z 748.539,A 0.000,B 0.000,C 90.000,E1 312.933} C_DIS
LIN {X 0.050,Y -685.382,Z 748.533,A 0.000,B 0.000,C 90.000,E1 312.000} C_DIS
LIN {X 0.467,Y -688.199,Z 748.526,A 0.000,B 0.000,C 90.000,E1 310.539} C_DIS
LIN {X -0.174,Y -689.736,Z 748.520,A 0.000,B 0.000,C 90.000,E1 309.644} C_DIS
LIN {X 0.110,Y -690.770,Z 748.516,A 0.000,B 0.000,C 90.000,E1 308.910} C_DIS
LIN {X -0.260,Y -692.605,Z 748.508,A 0.000,B 0.000,C 90.000,E1 307.523} C_DIS
LIN {X -0.309,Y -693.663,Z 748.503,A 0.000,B 0.000,C 90.000,E1 306.583} C_DIS
LIN {X -0.088,Y -694.953,Z 748.495,A 0.000,B 0.000,C 90.000,E1 305.152} C_DIS
LIN {X -0.293,Y -695.916,Z 748.489,A 0.000,B 0.000,C 90.000,E1 303.992} C_DIS
LIN {X -0.199,Y -697.213,Z 748.480,A 0.000,B 0.000,C 90.000,E1 302.339} C_DIS
LIN {X -0.117,Y -698.277,Z 748.472,A 0.000,B 0.000,C 90.000,E1 300.924} C_DIS
LIN {X 0.056,Y -698.680,Z 748.468,A 0.000,B 0.000,C 90.000,E1 300.207} C_DIS
LIN {X 0.158,Y -699.073,Z 748.461,A 0.000,B 0.000,C 90.000,E1 299.027} C_DIS
LIN {X 0.185,Y -699.592,Z 748.452,A 0.000,B 0.000,C 90.000,E1 297.385} C_DIS
LIN {X 0.123,Y -700.534,Z 748.441,A 0.000,B 0.000,C 90.000,E1 295.283} C_DIS
LIN {X 0.031,Y -700.611,Z 748.438,A 0.000,B 0.000,C 90.000,E1 294.823} C_DIS
LIN {X 0.010,Y -700.552,Z 748.437,A 0.000,B 0.000,C 90.000,E1 294.591} C_DIS
LIN {X -0.086,Y -699.788,Z 748.434,A 0.000,B 0.000,C 90.000,E1 294.131} C_DIS
LIN {X -0.102,Y -699.131,Z 748.433,A 0.000,B 0.000,C 90.000,E1 293.898} C_DIS
LIN {X 0.295,Y -697.164,Z 748.431,A 0.000,B 0.000,C 90.000,E1 293.515} C_DIS
LIN {X -0.362,Y -695.599,Z 748.430,A 0.000,B 0.000,C 90.000,E1 293.334} C_DIS
LIN {X -0.234,Y -694.497,Z 748.429,A 0.000,B 0.000,C 90.000,E1 293.206} C_DIS
LIN {X -0.108,Y -692.814,Z 748.428,A 0.000,B 0.000,C 90.000,E1 293.078} C_DIS
LIN {X -0.110,Y -685.748,Z 748.426,A 0.000,B 0.000,C 90.000,E1 292.717} C_DIS
LIN {X -0.184,Y -683.264,Z 748.426,A 0.000,B 0.000,C 90.000,E1 292.642} C_DIS
LIN {X -0.405,Y -674.878,Z 748.425,A 0.000,B 0.000,C 90.000,E1 292.461} C_DIS
LIN {X -0.099,Y -667.726,Z 748.424,A 0.000,B 0.000,C 90.000,E1 292.333} C_DIS
LIN {X 0.070,Y -658.397,Z 748.423,A 0.000,B 0.000,C 90.000,E1 292.206} C_DIS
LIN {X -0.196,Y -648.041,Z 748.423,A 0.000,B 0.000,C 90.000,E1 292.078} C_DIS
LIN {X -0.180,Y -638.336,Z 748.422,A 0.000,B 0.000,C 90.000,E1 291.897} C_DIS
LIN {X 0.030,Y -628.509,Z 748.420,A 0.000,B 0.000,C 90.000,E1 291.663} C_DIS
LIN {X 0.143,Y -611.196,Z 748.418,A 0.000,B 0.000,C 90.000,E1 291.227} C_DIS
LIN {X 0.090,Y -574.674,Z 748.412,A 0.000,B 0.000,C 90.000,E1 290.194} C_DIS
LIN {X 0.182,Y -567.233,Z 748.411,A 0.000,B 0.000,C 90.000,E1 289.993} C_DIS
LIN {X 0.171,Y -562.096,Z 748.410,A 0.000,B 0.000,C 90.000,E1 289.812} C_DIS
LIN {X 0.092,Y -560.647,Z 748.410,A 0.000,B 0.000,C 90.000,E1 289.758} C_DIS
LIN {X -0.179,Y -556.957,Z 748.409,A 0.000,B 0.000,C 90.000,E1 289.577} C_DIS
LIN {X 0.137,Y -555.770,Z 748.408,A 0.000,B 0.000,C 90.000,E1 289.396} C_DIS
LIN {X 0.095,Y -555.758,Z 748.408,A 0.000,B 0.000,C 90.000,E1 289.396} C_DIS
LIN {X 0.091,Y -555.103,Z 748.406,A 0.000,B 0.000,C 90.000,E1 289.087} C_DIS
LIN {X -0.035,Y -554.703,Z 748.403,A 0.000,B 0.000,C 90.000,E1 288.489} C_DIS
LIN {X 0.111,Y -554.479,Z 748.398,A 0.000,B 0.000,C 90.000,E1 287.638} C_DIS
LIN {X -0.059,Y -553.971,Z 748.390,A 0.000,B 0.000,C 90.000,E1 286.260} C_DIS
LIN {X -0.008,Y -553.247,Z 748.380,A 0.000,B 0.000,C 90.000,E1 284.300} C_DIS
LIN {X 0.184,Y -552.764,Z 748.372,A 0.000,B 0.000,C 90.000,E1 282.883} C_DIS
LIN {X -0.177,Y -552.209,Z 748.362,A 0.000,B 0.000,C 90.000,E1 281.243} C_DIS
LIN {X 0.197,Y -551.867,Z 748.356,A 0.000,B 0.000,C 90.000,E1 280.084} C_DIS
LIN {X 0.148,Y -551.262,Z 748.348,A 0.000,B 0.000,C 90.000,E1 278.690} C_DIS
LIN {X 0.222,Y -550.350,Z 748.338,A 0.000,B 0.000,C 90.000,E1 276.720} C_DIS
LIN {X -0.039,Y -549.829,Z 748.331,A 0.000,B 0.000,C 90.000,E1 275.625} C_DIS
LIN {X -0.181,Y -548.853,Z 748.322,A 0.000,B 0.000,C 90.000,E1 273.955} C_DIS
LIN {X 0.131,Y -547.974,Z 748.313,A 0.000,B 0.000,C 90.000,E1 272.236} C_DIS
LIN {X -0.119,Y -547.119,Z 748.303,A 0.000,B 0.000,C 90.000,E1 270.573} C_DIS
LIN {X 0.104,Y -546.224,Z 748.295,A 0.000,B 0.000,C 90.000,E1 269.141} C_DIS
LIN {X -0.115,Y -544.727,Z 748.283,A 0.000,B 0.000,C 90.000,E1 266.906} C_DIS
LIN {X 0.103,Y -543.866,Z 748.275,A 0.000,B 0.000,C 90.000,E1 265.469} C_DIS
LIN {X -0.232,Y -542.878,Z 748.267,A 0.000,B 0.000,C 90.000,E1 264.090} C_DIS
LIN {X 0.001,Y -542.083,Z 748.261,A 0.000,B 0.000,C 90.000,E1 262.932} C_DIS
LIN {X -0.231,Y -540.664,Z 748.251,A 0.000,B 0.000,C 90.000,E1 261.254} C_DIS
LIN {X 0.051,Y -539.488,Z 748.243,A 0.000,B 0.000,C 90.000,E1 259.803} C_DIS
LIN {X -0.165,Y -538.100,Z 748.234,A 0.000,B 0.000,C 90.000,E1 258.117} C_DIS
LIN {X 0.209,Y -537.111,Z 748.228,A 0.000,B 0.000,C 90.000,E1 256.937} C_DIS
LIN {X -0.076,Y -536.094,Z 748.221,A 0.000,B 0.000,C 90.000,E1 255.825} C_DIS
LIN {X -0.109,Y -534.854,Z 748.215,A 0.000,B 0.000,C 90.000,E1 254.685} C_DIS
LIN {X -0.256,Y -533.278,Z 748.207,A 0.000,B 0.000,C 90.000,E1 253.268} C_DIS
LIN {X 0.080,Y -531.078,Z 748.196,A 0.000,B 0.000,C 90.000,E1 251.221} C_DIS
LIN {X -0.219,Y -530.349,Z 748.193,A 0.000,B 0.000,C 90.000,E1 250.678} C_DIS
LIN {X 0.029,Y -528.404,Z 748.185,A 0.000,B 0.000,C 90.000,E1 249.209} C_DIS
LIN {X -0.252,Y -526.370,Z 748.177,A 0.000,B 0.000,C 90.000,E1 247.794} C_DIS
LIN {X -0.202,Y -523.744,Z 748.167,A 0.000,B 0.000,C 90.000,E1 246.049} C_DIS
LIN {X -0.147,Y -521.398,Z 748.159,A 0.000,B 0.000,C 90.000,E1 244.588} C_DIS
LIN {X 0.194,Y -519.481,Z 748.152,A 0.000,B 0.000,C 90.000,E1 243.384} C_DIS
LIN {X 0.036,Y -517.375,Z 748.146,A 0.000,B 0.000,C 90.000,E1 242.231} C_DIS
LIN {X -0.254,Y -514.542,Z 748.138,A 0.000,B 0.000,C 90.000,E1 240.795} C_DIS
LIN {X 0.102,Y -511.687,Z 748.129,A 0.000,B 0.000,C 90.000,E1 239.282} C_DIS
LIN {X 0.227,Y -508.805,Z 748.121,A 0.000,B 0.000,C 90.000,E1 237.788} C_DIS
LIN {X 0.083,Y -506.967,Z 748.116,A 0.000,B 0.000,C 90.000,E1 236.914} C_DIS
LIN {X 0.090,Y -504.294,Z 748.110,A 0.000,B 0.000,C 90.000,E1 235.722} C_DIS
LIN {X -0.113,Y -502.241,Z 748.105,A 0.000,B 0.000,C 90.000,E1 234.848} C_DIS
LIN {X 0.238,Y -500.115,Z 748.100,A 0.000,B 0.000,C 90.000,E1 233.909} C_DIS
LIN {X -0.129,Y -497.881,Z 748.095,A 0.000,B 0.000,C 90.000,E1 233.050} C_DIS
LIN {X 0.044,Y -494.796,Z 748.088,A 0.000,B 0.000,C 90.000,E1 231.823} C_DIS
LIN {X 0.161,Y -491.823,Z 748.081,A 0.000,B 0.000,C 90.000,E1 230.598} C_DIS
LIN {X 0.130,Y -486.138,Z 748.068,A 0.000,B 0.000,C 90.000,E1 228.162} C_DIS
LIN {X -0.027,Y -482.131,Z 748.057,A 0.000,B 0.000,C 90.000,E1 226.338} C_DIS
LIN {X -0.270,Y -478.212,Z 748.047,A 0.000,B 0.000,C 90.000,E1 224.514} C_DIS
LIN {X -0.033,Y -474.906,Z 748.039,A 0.000,B 0.000,C 90.000,E1 222.933} C_DIS
LIN {X 0.041,Y -472.255,Z 748.032,A 0.000,B 0.000,C 90.000,E1 221.676} C_DIS
LIN {X -0.039,Y -468.029,Z 748.021,A 0.000,B 0.000,C 90.000,E1 219.806} C_DIS
LIN {X -0.094,Y -463.274,Z 748.009,A 0.000,B 0.000,C 90.000,E1 217.604} C_DIS
LIN {X 0.187,Y -457.964,Z 747.995,A 0.000,B 0.000,C 90.000,E1 215.025} C_DIS
LIN {X -0.027,Y -454.739,Z 747.986,A 0.000,B 0.000,C 90.000,E1 213.452} C_DIS
LIN {X -0.057,Y -451.667,Z 747.977,A 0.000,B 0.000,C 90.000,E1 211.848} C_DIS
LIN {X -0.167,Y -448.074,Z 747.966,A 0.000,B 0.000,C 90.000,E1 209.922} C_DIS
LIN {X -0.099,Y -445.647,Z 747.959,A 0.000,B 0.000,C 90.000,E1 208.615} C_DIS
LIN {X -0.071,Y -443.275,Z 747.952,A 0.000,B 0.000,C 90.000,E1 207.308} C_DIS
LIN {X -0.044,Y -440.217,Z 747.943,A 0.000,B 0.000,C 90.000,E1 205.668} C_DIS
LIN {X -0.065,Y -437.136,Z 747.933,A 0.000,B 0.000,C 90.000,E1 204.027} C_DIS
LIN {X 0.073,Y -433.407,Z 747.922,A 0.000,B 0.000,C 90.000,E1 202.025} C_DIS
LIN {X -0.055,Y -431.549,Z 747.917,A 0.000,B 0.000,C 90.000,E1 201.046} C_DIS
LIN {X -0.165,Y -427.151,Z 747.904,A 0.000,B 0.000,C 90.000,E1 198.725} C_DIS
LIN {X 0.099,Y -424.610,Z 747.896,A 0.000,B 0.000,C 90.000,E1 197.347} C_DIS
LIN {X -0.245,Y -420.645,Z 747.885,A 0.000,B 0.000,C 90.000,E1 195.371} C_DIS
LIN {X 0.158,Y -416.250,Z 747.872,A 0.000,B 0.000,C 90.000,E1 192.939} C_DIS
LIN {X 0.075,Y -413.238,Z 747.863,A 0.000,B 0.000,C 90.000,E1 191.243} C_DIS
LIN {X -0.111,Y -409.741,Z 747.851,A 0.000,B 0.000,C 90.000,E1 189.208} C_DIS
LIN {X -0.012,Y -405.160,Z 747.836,A 0.000,B 0.000,C 90.000,E1 186.429} C_DIS
LIN {X -0.151,Y -401.481,Z 747.822,A 0.000,B 0.000,C 90.000,E1 184.012} C_DIS
LIN {X -0.049,Y -398.058,Z 747.809,A 0.000,B 0.000,C 90.000,E1 181.547} C_DIS
LIN {X -0.188,Y -394.374,Z 747.791,A 0.000,B 0.000,C 90.000,E1 178.396} C_DIS
LIN {X -0.121,Y -392.474,Z 747.781,A 0.000,B 0.000,C 90.000,E1 176.617} C_DIS
LIN {X 0.152,Y -390.193,Z 747.767,A 0.000,B 0.000,C 90.000,E1 174.090} C_DIS
LIN {X 0.184,Y -387.691,Z 747.744,A 0.000,B 0.000,C 90.000,E1 169.803} C_DIS
LIN {X -0.125,Y -386.711,Z 747.732,A 0.000,B 0.000,C 90.000,E1 167.701} C_DIS
LIN {X 0.087,Y -385.812,Z 747.720,A 0.000,B 0.000,C 90.000,E1 165.519} C_DIS
LIN {X -0.070,Y -384.975,Z 747.704,A 0.000,B 0.000,C 90.000,E1 162.670} C_DIS
LIN {X 0.059,Y -384.389,Z 747.690,A 0.000,B 0.000,C 90.000,E1 160.134} C_DIS
LIN {X 0.061,Y -384.047,Z 747.678,A 0.000,B 0.000,C 90.000,E1 157.975} C_DIS
LIN {X -0.137,Y -383.822,Z 747.664,A 0.000,B 0.000,C 90.000,E1 155.485} C_DIS
LIN {X -0.028,Y -386.625,Z 747.622,A 0.000,B 0.000,C 90.000,E1 147.916} C_DIS
LIN {X -0.150,Y -387.760,Z 747.614,A 0.000,B 0.000,C 90.000,E1 146.501} C_DIS
LIN {X 0.081,Y -390.150,Z 747.602,A 0.000,B 0.000,C 90.000,E1 144.322} C_DIS
LIN {X -0.096,Y -392.049,Z 747.594,A 0.000,B 0.000,C 90.000,E1 142.924} C_DIS
LIN {X -0.013,Y -394.724,Z 747.586,A 0.000,B 0.000,C 90.000,E1 141.492} C_DIS
LIN {X -0.141,Y -396.375,Z 747.582,A 0.000,B 0.000,C 90.000,E1 140.803} C_DIS
LIN {X 0.069,Y -398.470,Z 747.578,A 0.000,B 0.000,C 90.000,E1 140.070} C_DIS
LIN {X 0.063,Y -401.248,Z 747.574,A 0.000,B 0.000,C 90.000,E1 139.380} C_DIS
LIN {X -0.144,Y -403.226,Z 747.572,A 0.000,B 0.000,C 90.000,E1 139.013} C_DIS
LIN {X 0.060,Y -406.952,Z 747.569,A 0.000,B 0.000,C 90.000,E1 138.405} C_DIS
LIN {X 0.115,Y -410.998,Z 747.566,A 0.000,B 0.000,C 90.000,E1 137.877} C_DIS
LIN {X -0.195,Y -428.003,Z 747.556,A 0.000,B 0.000,C 90.000,E1 136.134} C_DIS
